// TwinCAT 3 PLC project tc_project_app
// ProgramVersion: 3.1.4023.0
// libraries:
//   Get_Nc_Error_Texts_and_descriptions, * (Beckhoff Automation GmbH & Co. KG)
//   Tc2_EtherCAT, * (Beckhoff Automation GmbH)
//   Tc2_MC2, * (Beckhoff Automation GmbH)
//   Tc2_Standard, * (Beckhoff Automation GmbH)
//   Tc2_SUPS, * (Beckhoff Automation GmbH)
//   Tc2_System, * (Beckhoff Automation GmbH)
//   Tc2_Utilities, * (Beckhoff Automation GmbH)
//   Tc3_MC2_AdvancedHoming, * (Beckhoff Automation GmbH)
//   Tc3_Module, * (Beckhoff Automation GmbH)
//   VisuDialogs, * (System)
//   Tc2_Math,3.3.1.0,Beckhoff Automation GmbH
//   VisuSymbols,3.5.10.0,System
// project tree:
//   DUTs/ E_Beamline.TcDUT, E_ResetZero.TcDUT, stFaultType.TcDUT, E_LightShutterSystemStates.TcDUT, E_SeqRangePosStates.TcDUT, E_NeutronFactoryStates.TcDUT, ST_LightShutter.TcDUT
//   / GlobalTextList.TcGTLO, PlcTask.TcTTO, PlcTaskCom.TcTTO, Visualization Manager.TcVMO (not stored)
//   GVLs/ GVL_APP.TcGVL
//   POUs/Application_Specific/Applications/ Application_Template.TcPOU, FB_ResetZero.TcPOU, HomeStepBlockDetection.TcPOU, NeutronFactoryStates.TcPOU, LightShutterSystemStates.TcPOU, SeqRangePos.TcPOU
//   POUs/Application_Specific/Axes/ Axis_Template.TcPOU, Pneumatics_Template.TcPOU
//   POUs/ MAIN.TcPOU
//   tc_mca_std_lib/DUTs/ E_AxisParameters.TcTLEO (not stored), E_HomingRoutines.TcTLEO (not stored), E_AxisParameters.TcTLEO (not stored), E_MotorTypeClass.TcDUT (not stored), E_EncoderTypeClass.TcDUT (not stored), E_HomeSwitchTypeClass.TcDUT (not stored), E_RestorePosition.TcDUT (not stored), E_SlitPairStates.TcDUT (not stored), ST_AxisConfig.TcDUT (not stored), ST_StepBlockConfig.TcDUT (not stored), ST_AxisControl.TcDUT (not stored), E_MotionFunctions.TcDUT (not stored), ST_AxisDescription.TcDUT (not stored), ST_AxisError.TcDUT (not stored), ST_AxisInputs.TcDUT (not stored), ST_AxisPersistent.TcDUT (not stored), ST_GearAxis.TcDUT (not stored), ST_AxisStatus.TcDUT (not stored), ST_AxisStruct.TcDUT (not stored)
//   tc_mca_std_lib/DUTs/Pneumatics/ E_PneumaticAxisErrors.TcDUT (not stored), E_PneumaticMode.TcDUT (not stored), ST_PneumaticAxisControl.TcDUT (not stored), ST_PneumaticAxisConfig.TcDUT (not stored), ST_PneumaticAxisInputs.TcDUT (not stored), ST_PneumaticAxisOutputs.TcDUT (not stored), ST_PneumaticAxisStatus.TcDUT (not stored), ST_PneumaticAxisStruct.TcDUT (not stored)
//   tc_mca_std_lib/GVLs/ GVL.TcGVL (not stored)
//   tc_mca_std_lib/POUs/Motion/ FB_Axis.TcPOU (not stored), FB_SlitPair.TcPOU (not stored)
//   tc_mca_std_lib/POUs/Motion/Homing/ FB_Homing.TcPOU (not stored)
//   tc_mca_std_lib/POUs/Pneumatics/ FB_PneumaticAxis.TcPOU (not stored)
//   tc_mca_std_lib/VISUs/ languageSupport.TcTLO (not stored), MainVisu.TcVIS (not stored), PneumaticsVisu.TcVIS (not stored), visuTextLinks.TcTLO (not stored)
//   tc_pils/tc_pils_app_specific/GVLs/ GVL_PILS.TcGVL
//   tc_pils/tc_pils_app_specific/POUs/ PILS_DEVICES.TcPOU
//   tc_pils/tc_pils_generic/DUTs/ E_Permission.TcDUT (not stored), E_PILS_ParamControl.TcDUT (not stored), E_PILS_ParamControlCmd.TcDUT (not stored), E_PILS_State.TcDUT (not stored), ST_1201.TcDUT (not stored), ST_1202.TcDUT (not stored), ST_1204.TcDUT (not stored), ST_1602.TcDUT (not stored), ST_5008.TcDUT (not stored), ST_5010.TcDUT (not stored), ST_AxisParameters.TcDUT (not stored), ST_DeviceInfo.TcDUT (not stored), ST_Indexer.TcDUT (not stored), ST_Indexer_InfoTyp0.TcDUT (not stored), ST_ParamOutput.TcDUT (not stored), U_IndexerData.TcDUT (not stored)
//   tc_pils/tc_pils_generic/POUs/ COMM.TcPOU (not stored)
//   tc_pils/tc_pils_generic/POUs/PILS_device_types/ FB_5010_Axis.TcPOU (not stored)
//   VISUs/ AcceleratorStates.TcVIS, languageTable.TcTLO, StepBlockDetection.TcVIS
// real-time tasks:
//   TASK PlcTask: cycle T#10ms, priority 10, ADS port 351
//   TASK PlcTaskCom: cycle T#2ms, priority 5, ADS port 350
// motion (NC):
//   TASK NC-Task 1 SAF: cycle T#2ms, priority 4, ADS port 501
//   TASK NC-Task 1 SVB: cycle T#10ms, priority 8, ADS port 511
//   AXIS Axis 1 (id 1)
//     Dynamic: AccelerationMaximum=1500, DecelerationMaximum=1500, Acceleration=50, Deceleration=50, Jerk=1000
//     Velo: RefSearch=10, RefSync=10, SlowManual=10, FastManual=15, Maximum=500
//     PositionAreaControl: Range=0.5
//     TargetPosControl: Range=0.5, Time=0.2
//     OtherSettings: AllowMotionCmdToSlave=true, PulseDistancePos=10, PulseDistanceNeg=10
//     encoder EncType=5
//       EncPara: ScaleFactorNumerator=60, ScaleFactorDenominator=4096, Inverse=true, ReferenceSystem=1
//         SoftEndMinControl: Range=1
//         SoftEndMaxControl: Range=500000
//         Inc: RefSoftSyncMask=#x0000ffff
//     drive DrvType=24
//       Analog: VeloReferenz=600, TorqueSetpointScale=10, ScaleFactorActTorque=0.1
//       TimeComp: TaskDelayCycles=1
//     controller CtrType=1
//       CtrPara: PriorControlFactor=1
//         PosDiffControl: Range=100
//         Observer: BandWidth=20
//   AXIS Axis 2 (id 2)
//     Dynamic: AccelerationMaximum=1500, DecelerationMaximum=1500, Acceleration=50, Deceleration=50, Jerk=1000
//     Velo: RefSearch=10, RefSync=10, SlowManual=10, FastManual=15, Maximum=500
//     PositionAreaControl: Range=0.5
//     TargetPosControl: Range=0.5, Time=0.2
//     OtherSettings: AllowMotionCmdToSlave=true, PulseDistancePos=10, PulseDistanceNeg=10
//     encoder EncType=5
//       EncPara: ScaleFactorNumerator=60, ScaleFactorDenominator=4096, Inverse=true, MaxCount=#xffffffff, ReferenceSystem=1
//         SoftEndMinControl: Range=1
//         SoftEndMaxControl: Range=500000
//         Inc: RefSoftSyncMask=#x0000ffff
//     drive DrvType=24
//       Analog: VeloReferenz=600, TorqueSetpointScale=10, ScaleFactorActTorque=0.1
//       TimeComp: TaskDelayCycles=1
//     controller CtrType=1
//       CtrPara: PriorControlFactor=1
//         PosDiffControl: Range=100
//         Observer: BandWidth=20
//   AXIS Axis 3 (id 3)
//     Dynamic: Acceleration=3439.33, Deceleration=3439.33, Jerk=10318
//     Velo: RefSearch=22.9288618666667, RefSync=22.9288618666667, SlowManual=114.644309333333, FastManual=687.865856, Fast=2292.88618666667, Maximum=2292.89
//     OtherSettings: AllowMotionCmdToSlave=true
//     encoder EncType=19
//       EncPara: ScaleFactorNumerator=104.8576, ScaleFactorDenominator=1048576, MaxCount=#xffffffff
//     drive DrvType=16
//       DrvPara: MaxCount=#xffffffff, DriveControlDWord=#x00020000
//         Analog: VeloReferenz=2522.17480533333, VeloScale=32, TorqueSetpointScale=10, ScaleFactorActTorque=0.1
//         TimeComp: TaskDelayCycles=1
//     controller CtrType=1
//       CtrPara: PriorControlFactor=1
//         PosDiffControl: Enable=false
//         Observer: BandWidth=20
// I/O:
//   DEVICE Device 1 (EtherCAT), AmsNetId 5.65.73.226.2.1
//     Term 1 (EK1200) [EK1200-5000 EtherCAT Power supply (2A E-Bus)]
//       Term 2 (EL1808) [EL1808 8Ch. Dig. Input 24V, 3ms]
//       Term 3 (EL2819) [EL2819 16Ch. Dig. Output 24V, 0,5A, Diagnostic]
//       Term 4 (EL5002) [EL5002 2Ch. SSI Encoder]
//       Term 5 (EL2014) [EL2014 4Ch. Dig. Output 24V, 0,5A, Diagnostic]
//       Term 6 (EL7041-0052) [EL7041-0052 1Ch. Stepper motor output stage (50V, 5A)]
//       Term 7 (EL7041-0052) [EL7041-0052 1Ch. Stepper motor output stage (50V, 5A)]
//       Term 8 (EL3204) [EL3204 4Ch. Ana. Input PT100 (RTD)]
//       Term 18 (EL7201) [EL7201 1Ch. MDP742 Servo motor output stage (50V, 4A)]
//       Term 9 (EL9011) [EL9011 End Terminal]
//   DEVICE Device 4 (COM Port)
// variable links:
//   (this object) <-> Device 1 (EtherCAT)/Term 1 (EK1200)/Term 4 (EL5002)
//     Enc/Inputs/In/nDataIn1 <-> SSI Inputs Channel 1/Counter value
//     Enc/Inputs/In/nDataIn1 <-> SSI Inputs Channel 2/Counter value
//     Enc/Inputs/In/nState1 <-> SSI Inputs Channel 1/Data error
//     Enc/Inputs/In/nState1 <-> SSI Inputs Channel 2/Data error
//     Enc/Inputs/In/nState1 @bit 3 <-> SSI Inputs Channel 1/Data mismatch
//     Enc/Inputs/In/nState1 @bit 3 <-> SSI Inputs Channel 2/Data mismatch
//     Enc/Inputs/In/nState1 @bit 1 <-> SSI Inputs Channel 1/Frame error
//     Enc/Inputs/In/nState1 @bit 1 <-> SSI Inputs Channel 2/Frame error
//     Enc/Inputs/In/nState1 @bit 2 <-> SSI Inputs Channel 1/Power failure
//     Enc/Inputs/In/nState1 @bit 2 <-> SSI Inputs Channel 2/Power failure
//     Enc/Inputs/In/nState2 @bit 5 <-> SSI Inputs Channel 1/Sync error
//     Enc/Inputs/In/nState2 @bit 5 <-> SSI Inputs Channel 2/Sync error
//     Enc/Inputs/In/nState2 @bit 6 <-> SSI Inputs Channel 1/TxPDO State
//     Enc/Inputs/In/nState2 @bit 6 <-> SSI Inputs Channel 2/TxPDO State
//     Enc/Inputs/In/nState2 @bit 7 <-> SSI Inputs Channel 1/TxPDO Toggle
//     Enc/Inputs/In/nState2 @bit 7 <-> SSI Inputs Channel 2/TxPDO Toggle
//     Enc/Inputs/In/nState4 @bit 1 <-> WcState/InputToggle
//     Enc/Inputs/In/nState4 <-> WcState/WcState
//   (this object) <-> Device 1 (EtherCAT)/Term 1 (EK1200)/Term 6 (EL7041-0052)
//     Drive/Inputs/In/nState1 @bit 3 <-> STM Status/Error
//     Drive/Inputs/In/nState1 @bit 5 <-> STM Status/Moving negative
//     Drive/Inputs/In/nState1 @bit 4 <-> STM Status/Moving positive
//     Drive/Inputs/In/nState1 @bit 1 <-> STM Status/Ready
//     Drive/Inputs/In/nState1 <-> STM Status/Ready to enable
//     Drive/Inputs/In/nState1 @bit 6 <-> STM Status/Torque reduced
//     Drive/Inputs/In/nState1 @bit 2 <-> STM Status/Warning
//     Drive/Inputs/In/nState2 @bit 3 <-> STM Status/Digital input 1
//     Drive/Inputs/In/nState2 @bit 4 <-> STM Status/Digital input 2
//     Drive/Inputs/In/nState2 @bit 5 <-> STM Status/Sync error
//     Drive/Inputs/In/nState2 @bit 7 <-> STM Status/TxPDO Toggle
//     Drive/Inputs/In/nState4 @bit 1 <-> WcState/InputToggle
//     Drive/Inputs/In/nState4 <-> WcState/WcState
//     Drive/Outputs/Out/nCtrl1 <-> STM Control/Enable
//     Drive/Outputs/Out/nCtrl1 @bit 2 <-> STM Control/Reduce torque
//     Drive/Outputs/Out/nCtrl1 @bit 1 <-> STM Control/Reset
//     Drive/Outputs/Out/nDataOut2[0] <-> STM Velocity/Velocity
//   (this object) <-> Device 1 (EtherCAT)/Term 1 (EK1200)/Term 7 (EL7041-0052)
//     Drive/Inputs/In/nState1 @bit 3 <-> STM Status/Status/Error
//     Drive/Inputs/In/nState1 @bit 5 <-> STM Status/Status/Moving negative
//     Drive/Inputs/In/nState1 @bit 4 <-> STM Status/Status/Moving positive
//     Drive/Inputs/In/nState1 @bit 1 <-> STM Status/Status/Ready
//     Drive/Inputs/In/nState1 <-> STM Status/Status/Ready to enable
//     Drive/Inputs/In/nState1 @bit 6 <-> STM Status/Status/Torque reduced
//     Drive/Inputs/In/nState1 @bit 2 <-> STM Status/Status/Warning
//     Drive/Inputs/In/nState2 @bit 3 <-> STM Status/Status/Digital input 1
//     Drive/Inputs/In/nState2 @bit 4 <-> STM Status/Status/Digital input 2
//     Drive/Inputs/In/nState2 @bit 5 <-> STM Status/Status/Sync error
//     Drive/Inputs/In/nState2 @bit 7 <-> STM Status/Status/TxPDO Toggle
//     Drive/Inputs/In/nState4 @bit 1 <-> WcState/InputToggle
//     Drive/Inputs/In/nState4 <-> WcState/WcState
//     Drive/Outputs/Out/nCtrl1 <-> STM Control/Control/Enable
//     Drive/Outputs/Out/nCtrl1 @bit 2 <-> STM Control/Control/Reduce torque
//     Drive/Outputs/Out/nCtrl1 @bit 1 <-> STM Control/Control/Reset
//     Drive/Outputs/Out/nDataOut2[0] <-> STM Velocity/Velocity
//   (this object) <-> Device 1 (EtherCAT)/Term 1 (EK1200)/Term 18 (EL7201)
//     Drive/Inputs/In/nDcOutputTime <-> InfoData/DcOutputShift
//     Drive/Inputs/In/nState1 <-> DRV Statusword/Statusword
//     Drive/Inputs/In/nState2 <-> DRV Statusword/Statusword @bit 8
//     Drive/Inputs/In/nState4 @bit 1 <-> WcState/InputToggle
//     Drive/Inputs/In/nState4 <-> WcState/WcState
//     Drive/Outputs/Out/nCtrl1 <-> DRV Controlword/Controlword
//     Drive/Outputs/Out/nCtrl2 <-> DRV Controlword/Controlword @bit 8
//     Drive/Outputs/Out/nDataOut2 <-> DRV Target velocity/Target velocity
//     Enc/Inputs/In/nDataIn1 <-> FB Position/Position
//     Enc/Inputs/In/nDcInputTime <-> InfoData/DcInputShift
//     Enc/Inputs/In/nState4 @bit 1 <-> WcState/InputToggle
//     Enc/Inputs/In/nState4 <-> WcState/WcState
//   tc_project_app Instance <-> Device 1 (EtherCAT)/Term 1 (EK1200)/Term 2 (EL1808)
//     PlcTaskCom Inputs/GVL.astAxes[1].stInputs.bHomeSensor <-> Channel 3/Input
//     PlcTaskCom Inputs/GVL.astAxes[2].stInputs.bHomeSensor <-> Channel 7/Input
//     PlcTaskCom Inputs/GVL.astAxes[1].stInputs.bLimitBwd <-> Channel 2/Input
//     PlcTaskCom Inputs/GVL.astAxes[2].stInputs.bLimitBwd <-> Channel 6/Input
//     PlcTaskCom Inputs/GVL.astAxes[1].stInputs.bLimitFwd <-> Channel 1/Input
//     PlcTaskCom Inputs/GVL.astAxes[2].stInputs.bLimitFwd <-> Channel 5/Input
//   tc_project_app Instance <-> Device 1 (EtherCAT)/Term 1 (EK1200)/Term 3 (EL2819)
//     PlcTaskCom Outputs/Axis_Template.bPowerSwitchesAxis1 <-> DIG Outputs/Channel 1/Output
//     PlcTaskCom Outputs/Axis_Template.bPowerSwitchesAxis2 <-> DIG Outputs/Channel 5/Output
//   tc_project_app Instance <-> Device 1 (EtherCAT)/Term 1 (EK1200)/Term 5 (EL2014)
//     PlcTask Outputs/Axis_Template.bPowerEncAxis1 <-> DIG Outputs/Channel 1/Output
//     PlcTask Outputs/Axis_Template.bPowerEncAxis2 <-> DIG Outputs/Channel 2/Output
//   tc_project_app Instance <-> NC-Task 1 SAF/Axes/Axis 1
//     PlcTask Inputs/GVL.astAxes[1].Axis.NcToPlc <-> Outputs/ToPlc
//     PlcTask Outputs/GVL.astAxes[1].Axis.PlcToNc <-> Inputs/FromPlc
//   tc_project_app Instance <-> NC-Task 1 SAF/Axes/Axis 2
//     PlcTask Inputs/GVL.astAxes[2].Axis.NcToPlc <-> Outputs/ToPlc
//     PlcTask Outputs/GVL.astAxes[2].Axis.PlcToNc <-> Inputs/FromPlc
//   tc_project_app Instance <-> NC-Task 1 SAF/Axes/Axis 3
//     PlcTask Inputs/GVL.astAxes[3].Axis.NcToPlc <-> Outputs/ToPlc
//     PlcTask Outputs/GVL.astAxes[3].Axis.PlcToNc <-> Inputs/FromPlc

CONFIGURATION tc_project_app
    RESOURCE PLC ON TwinCAT3
        TASK PlcTask(INTERVAL := T#10ms, PRIORITY := 10);
        TASK PlcTaskCom(INTERVAL := T#2ms, PRIORITY := 5);
        PROGRAM MAIN WITH PlcTask : MAIN;
        PROGRAM COMM WITH PlcTaskCom : COMM;
    END_RESOURCE
END_CONFIGURATION

// ---- DUTs/E_Beamline.TcDUT
{attribute 'qualified_only'}
{attribute 'strict'}
TYPE E_Beamline :
(
    Miracles := 1,
	Heimdal
);
END_TYPE

// ---- DUTs/E_ResetZero.TcDUT
{attribute 'qualified_only'}
{attribute 'strict'}
TYPE E_ResetZero :
(
    INIT := 0,
	HOME_AXIS,
	FIND_POS_ONE,
	PREPARE_POS_ONE_X,
	RECORD_POS_ONE_X,
	PREPARE_POS_ONE_Y,
	RECORD_POS_ONE_Y,
	FIND_POS_TWO,
	POSITIONING
);
END_TYPE

// ---- DUTs/stFaultType.TcDUT
TYPE stFaultType :
	STRUCT
		sFaultType	:	STRING(255);
	END_STRUCT
END_TYPE

// ---- DUTs/E_LightShutterSystemStates.TcDUT
{attribute 'qualified_only'}
{attribute 'strict'}
TYPE E_LightShutterSystemStates :
(
    Init := 0,
	ClosedOff,
	ClosedStandby,
	Opening,
	Open,
	OpenToOpen,
	Adjusting,
	ResetZero,
	Closing,
	Maintenance,
	SinglePortMaintenance_ClosedStandby,
	SinglePortMaintenance_Opening,
	SinglePortMaintenance_Open,
	SinglePortMaintenance_Closing,
	LSS_Maintenance,
	Fault	
);
END_TYPE

// ---- DUTs/E_SeqRangePosStates.TcDUT
{attribute 'qualified_only'}
{attribute 'strict'}
TYPE E_SeqRangePosStates :
(
    INIT := 0,
    CHECK_HOME_STATUS,
    HOME_MOTOR,
    CHECK_HOME_COMPLETE,
    MOTOR_OPERATIONAL,
	POS_ZERO,
	POS_ONE,
	POS_TWO,
	POSITIONING,
    CLEAR_CALIBRATION,
    ERROR,
    ERROR_RESET_AXES,
    ERROR_RESET_CHECK
);
END_TYPE

// ---- DUTs/E_NeutronFactoryStates.TcDUT
{attribute 'qualified_only'}
{attribute 'strict'}
TYPE E_NeutronFactoryStates :
(
    Disabled := 0,
	Maintenance,
	StartUp,
	CoolingDown,
	NotConfirmedReady,
	ConfirmedReady	
);
END_TYPE

// ---- DUTs/ST_LightShutter.TcDUT
(*These are axis parameters that are set up during commissioning and
in theory don't neeed to be change as part of daily moving of axes.
For instance they may be changed due to poor parameter selection
or change of instrument configuration.*)
TYPE ST_LightShutter :
STRUCT
	//name? beamline nbr?
	// Are we also to store closed position?
    // Add status of switches?
	nbrOfPos : USINT; // 1 or 2 foxal points
	curPosNbr : USINT := 1;
	pos : ARRAY[1..2] OF LREAL := [0,0];
	
END_STRUCT
END_TYPE

// ---- GVLs/GVL_APP.TcGVL
{attribute 'qualified_only'}
VAR_GLOBAL
	aPosSwitch : ARRAY[1..GVL_APP.nAXIS_NUM, 1..2] OF BOOL;
END_VAR

VAR_GLOBAL CONSTANT
    nAXIS_NUM: UINT := 3; (*~ (OPC: 1 : available for OPC-clients)
                         (OPC_PROP[0005]: 1 : OPC_PROP_RIGHTS, here read only) *)
    nPNEUMATIC_AXIS_NUM: UINT := 0;
END_VAR

VAR_GLOBAL PERSISTENT
	aLightShutters : ARRAY[1..GVL_APP.nAXIS_NUM] OF ST_LightShutter;
END_VAR

// ---- tc_pils/tc_pils_app_specific/GVLs/GVL_PILS.TcGVL
  VAR_GLOBAL
    sPLCName: STRING[34] := 'Crate_026';
    sPLCVersion: STRING[34] := '0.9.3';
    sPLCAuthor1: STRING[34] := 'tc_lab_mcu026.git';
    sPLCAuthor2: STRING[34] := 'ESS Lund';

//PILS Devices
//First available memory area for PILS devices is 104. 64-99 is used by the indexer
//Run the python script "check_fix_gvl_pils.py" to check that the PILS devices have a correct memory allocation

    //Axis #1                  Pils-device typ
    stMotorM1       AT %MB104: ST_5010;
    fbMotorM1: FB_5010_Axis := (nPILSDeviceNumber := 1);
    stMotorM1Param: ST_AxisParameters := (eMicrostepsPermission := E_Permission.eHidden,
                                          eResolutionPermission := E_Permission.eHidden,
                                          eAccelerationPermission := E_Permission.eWrite,
                                          eHomePositionPermission := E_Permission.eWrite,
                                          eHomingVelocityPermission := E_Permission.eWrite,
                                          eLagErrorPermission := E_Permission.eWrite,
                                          eTargetPositionWindowPermission := E_Permission.eWrite,
                                          eUserMaxPermission := E_Permission.eWrite,
                                          eUserMinPermission := E_Permission.eWrite,
                                          eVelocityPermission := E_Permission.eWrite,
                                          eSoftPosMinimumLimitEnablePermission := E_Permission.eWrite,
                                          eSoftPosMaximumLimitEnablePermission := E_Permission.eWrite,
                                          eHomeSequencePermission := E_Permission.eWrite,
                                          eEncoderScalingNumeratorPermission := E_Permission.eWrite,
                                          eEncoderScalingDenominatorPermission := E_Permission.eWrite,
                                          eMaximumVelocityPermission := E_Permission.eWrite);
										  
	//Axis #2                  Pils-device typ
    stMotorM2       AT %MB136: ST_5010;
    fbMotorM2: FB_5010_Axis := (nPILSDeviceNumber := 2);
    stMotorM2Param: ST_AxisParameters := (eMicrostepsPermission := E_Permission.eHidden,
                                          eResolutionPermission := E_Permission.eHidden,
                                          eAccelerationPermission := E_Permission.eWrite,
                                          eHomePositionPermission := E_Permission.eWrite,
                                          eHomingVelocityPermission := E_Permission.eWrite,
                                          eLagErrorPermission := E_Permission.eWrite,
                                          eTargetPositionWindowPermission := E_Permission.eWrite,
                                          eUserMaxPermission := E_Permission.eWrite,
                                          eUserMinPermission := E_Permission.eWrite,
                                          eVelocityPermission := E_Permission.eWrite,
                                          eSoftPosMinimumLimitEnablePermission := E_Permission.eWrite,
                                          eSoftPosMaximumLimitEnablePermission := E_Permission.eWrite,
                                          eHomeSequencePermission := E_Permission.eWrite,
                                          eEncoderScalingNumeratorPermission := E_Permission.eWrite,
                                          eEncoderScalingDenominatorPermission := E_Permission.eWrite,
                                          eMaximumVelocityPermission := E_Permission.eWrite);
										  
								
	stPowerSwitchesAxis1	AT %MB168: ST_1201;
	//fbMotorM2: FB_5010_Axis := (nPILSDeviceNumber := 2);
	//stPowerSwitchesAxis2	AT %MB170: ST_1201;
	stPowerSwitchesAxis2	AT %MB170: ST_1201;
	stPowerSwitchesAxis1Ctr AT %MB172: ST_1602;
	//stPowerSwitchesAxis2Ctr AT %MB176: ST_1602;
	

// Array of Devices
// Modify the array to fit the number of devices you have
// nUnit codes: mm = 16xfd04, degrees = 16x000C, Celsius =16x0009, Kelvin 16x0008

    astDevices: ARRAY [1..6] OF ST_DeviceInfo :=[ 									//axis specific.........generic
        (nTypCode := 16#5010, sName := 'M1 Lower', nOffset := 104, nUnit := 16#FD04, asAUX := [(''),(''),(''),(''),(''),(''),(''),(''),(''),(''),(''),(''),(''),(''),(''),(''),(''),('InterlockFwd'),('InterlockBwd'),('localMode'),('inTargetPos'),('homeSensor'),('notHomed'),('enabled')], nFlags := 1),
		(nTypCode := 16#5010, sName := 'M2 Higher', nOffset := 136, nUnit := 16#FD04, asAUX := [(''),(''),(''),(''),(''),(''),(''),(''),(''),(''),(''),(''),(''),(''),(''),(''),(''),('InterlockFwd'),('InterlockBwd'),('localMode'),('inTargetPos'),('homeSensor'),('notHomed'),('enabled')], nFlags := 1),
		(nTypCode := 16#1201, sName:= 'bPowerSwitchesAxis#1', nOffset := 168),
		(nTypCode := 16#1201, sName:= 'bPowerSwitchesAxis#2', nOffset := 170),
		(nTypCode := 16#1602, sName:= 'bPowerSwitchesAxisCtr#1', nOffset := 172)
		//(nTypCode := 16#1602, sName:= 'bPowerSwitchesAxisCtr#2', nOffset := 176)
		];
END_VAR

// ---- POUs/MAIN.TcPOU
PROGRAM MAIN
VAR
    sVersion: STRING := '1.0.0';
    afbAxes: ARRAY [1..GVL_APP.nAXIS_NUM] OF FB_Axis;
    afbPneumaticAxes: ARRAY [1..GVL_APP.nPNEUMATIC_AXIS_NUM] OF FB_PneumaticAxis;
    hmiAxisSelection: INT := 1; //Not possible to use local hmi variables for array indexes
    hmiPneumaticAxisSelection: INT := 1;
//Startup, Shutdown and UPS
    fbUPS: FB_S_UPS_CX51x0;
    eUpsMode: E_S_UPS_Mode := eSUPS_WrPersistData_Shutdown;
    eStartUp: (eColdStart, eReadAxisFeedbackType, eCheckReadDone, eExecuteRestore, eCheckRestore, eFinishRestore);
    bPositionRestoreDone: BOOL := FALSE;
    bRestoreExecute: BOOL := FALSE;
    bExecuteReadEncRefSys: BOOL := FALSE;
    nRetry: INT;
    iAxes : UINT; //index for for loops in Position recovery actions
    afbReadEncRefSys: ARRAY [1..GVL_APP.nAXIS_NUM] OF MC_ReadParameter;
    afbRestorePosition: ARRAY [1..GVL_APP.nAXIS_NUM] OF MC_SetPosition;
    fbGetDeviceIdentification: FB_GetDeviceIdentificationEx;
END_VAR

VAR PERSISTENT
    bRestoreOnStartup: BOOL;
END_VAR

POSITION_RECOVERY();
AXES();
PROG();

ACTION AXES:
//Get task index for Axes parameters initialization.
GVL.fbGetCurTaskIndex();

//Create an stAxisStruct for every axis in the project.
FOR GVL.iAxis := 1 TO GVL_APP.nAXIS_NUM DO
    afbAxes[GVL.iAxis](stAxisStruct := GVL.astAxes[GVL.iAxis]);
END_FOR

FOR GVL.iPneumaticAxis := 1 TO GVL_APP.nPNEUMATIC_AXIS_NUM DO
    afbPneumaticAxes[GVL.iPneumaticAxis](stPneumaticAxisStruct := GVL.astPneumaticAxes[GVL.iPneumaticAxis]);
END_FOR
END_ACTION

ACTION CHECK_UPS:
fbUPS(eUpsMode := eUpsMode);

IF eGlobalSUpsState = eSUPS_PowerFailure THEN
    //first cycle of powerfailure
    //execute code that should only be done once with each powerfailure, i.e. increase powerfailure counter
    bRestoreOnStartup := TRUE;
    STORE_PERSISTENT();
    RETURN;
ELSIF eGlobalSUpsState <> eSUPS_PowerOK THEN
    //next cycles of powerfailure
    //skip regular code execution for the remaining cycles of the powerfailure/writing of persistent data/quick shutdown...
    RETURN;
END_IF
END_ACTION

ACTION POSITION_RECOVERY:
fbGetDeviceIdentification(bExecute := TRUE);
IF (fbGetDeviceIdentification.stDevIdent.strHardwareSerialNo <> '0') THEN
    CHECK_UPS();
    RESTORE_POSITIONS();
END_IF
END_ACTION

ACTION PROG:
//Call the programs that are defined in the "Application Specific" folder.
//Create as many programs in that folder as axes and applications you have or need

//Axes program calls
Axis_Template();
Pneumatics_Template();

//Application program calls
Application_Template();
//SeqRangePos();
//NeutronFactoryStates();

//LightShutterSystemStates();
HomeStepBlockDetection();
END_ACTION

ACTION RESTORE_POSITIONS:
//This ACT will restore the position of an incremental axis on startup with the act position it read before losing power.
//It checks the type of axis, 0=incremental, and that the axis was stationary at shut down.
//Because 0 equates to incremental we also need to check that the data is valid, otherwise by default it would restore all axes.
//By default an axis will not restore the position unless it is set to opt-in, i.e. GVL.aAxes[iAxes].stConfig.eRestorePosition is non-zero.
//This needs to be initialised somewhere in TwinCAT code otherwise it will not be available at start up.
//A restore will only be performed on a loss of power, this code shouldn't make any changes on a reset cold, a rest origin or a download.
//There is a enum to allow for different types of restore modes, currently only one is implemented.
//0 'DontRestore'
//1 'RestoreWithoutHome' -restores the position using a set position fb and does not set the home bit in the axis struct.
//Note from Beckhoff: "A maximum of 1 MB persistent data can be reliably saved over the entire service life."

IF bRestoreOnStartup AND eGlobalSUpsState = eSUPS_PowerOK THEN
    bRestoreOnStartup := FALSE;
    bRestoreExecute := TRUE;
END_IF

//Upon startup bPositionRestoreDone will be set to FALSE, after successfully completing the following code it will be set TRUE
//and should stay TRUE for the rest of the time the PLC is operational, thus this routine should only be completed once.
IF bRestoreExecute AND NOT bPositionRestoreDone THEN
    //Cycle through function blocks that read the encoder reference system i.e. whether axis is incremental or absolute
    //Result stored in Value, 0=Inc 1=Abs, execute set during the case statement
    FOR iAxes := 1 TO GVL_APP.nAXIS_NUM DO
        afbReadEncRefSys[iAxes](
          Axis := GVL.astAxes[iAxes].Axis,
          Enable := bExecuteReadEncRefSys,
          ParameterNumber := MC_AxisParameter.AxisEncoderReferenceSystem,
          ReadMode := E_READMODE.READMODE_ONCE);
    END_FOR

    //Cycle through set position function blocks for each axis
    FOR iAxes := 1 TO GVL_APP.nAXIS_NUM DO
        afbRestorePosition[iAxes](
         Axis := GVL.astAxes[iAxes].Axis,
         Position := astAxesPersistent[iAxes].fPositionAtShutdown);
    END_FOR

    CASE eStartUp OF
        eColdStart:
        //First cycle of the PLC, do nothing just give one cycle for variables to initialise
            IF NOT bPositionRestoreDone THEN
                eStartUp := eReadAxisFeedbackType;
                nRetry := 0;
            END_IF

        eReadAxisFeedbackType:
        //Exectute the function blocks to read the encoder reference system (0=inc OR 1=ABS)
            bExecuteReadEncRefSys := TRUE;
            eStartUp := eCheckReadDone;

        eCheckReadDone:
        //Check the encoder reference system has been read for all axis -> if busy then continue with PLC cycle and check again next time.
        //If afbReadEncRefSys not started then go back a step.
        //If any axes result in an error the code will get stuck here, this happens if GVL_APP.nAXIS_NUM is not set correctly
            FOR iAxes := 1 TO GVL_APP.nAXIS_NUM DO
                IF afbReadEncRefSys[iAxes].Valid = FALSE THEN
                    IF afbReadEncRefSys[iAxes].Busy = TRUE THEN
                        //Exit MAIN.STARTUP Action and wait till next cycle, needs to cycle through whole program in order for data to update
                        RETURN;
                    ELSE
                        //Sometimes the code gets here and the afbReadEncRefSys[iAxes] misses the rising edge. If  the code gets here it means
                        //valid=FALSE and .busy=FALSE which indicateds the FB probably hasn't started and thus needs to see a rising edge.
                        //Set execute to low, Exit MAIN.STARTUP and go back a step in the CASE statement.
                        bExecuteReadEncRefSys := FALSE;
                        eStartUp := eReadAxisFeedbackType;
                        nRetry := nRetry + 1; //counter used for troubleshooting to see how many cycles it takes before afbReadEncRefSys function blocks are read correctly
                        RETURN;
                    END_IF
                END_IF
            END_FOR
            //If the code gets here all axes either have .valid=TRUE for all axes
            eStartUp := eExecuteRestore;

        eExecuteRestore:
        //Execute position restore by setting afbRestorePosition.execute = TRUE
            FOR iAxes := 1 TO GVL_APP.nAXIS_NUM DO
                IF afbReadEncRefSys[iAxes].Valid = TRUE AND afbReadEncRefSys[iAxes].Value = 0 AND NOT(astAxesPersistent[iAxes].bMovingAtShutdown) THEN
                    IF GVL.astAxes[iAxes].stConfig.eRestorePosition = E_RestorePosition.eRestoreWithoutHome THEN
                        afbRestorePosition[iAxes].Execute := TRUE;
                    END_IF
                END_IF
            END_FOR
            eStartUp := eCheckRestore;

        eCheckRestore:
        //Check the set position fbs are finished
        //Nothing actually happens if the restore is not done, the code just returns from here each cycle and the
        //bPositionRestoreDone will never get set to TRUE and will take up cycle time
            FOR iAxes := 1 TO GVL_APP.nAXIS_NUM DO
                IF afbReadEncRefSys[iAxes].Valid = TRUE AND afbReadEncRefSys[iAxes].Value = 0 AND NOT(astAxesPersistent[iAxes].bMovingAtShutdown) THEN
                    IF GVL.astAxes[iAxes].stConfig.eRestorePosition = E_RestorePosition.eRestoreWithoutHome THEN
                        IF NOT afbRestorePosition[iAxes].Done THEN
                            RETURN;
                        END_IF
                    END_IF
                END_IF
            END_FOR
            eStartUp := eFinishRestore;

        eFinishRestore:
        //Remove execute = TRUE for afbRestorePosition
            FOR iAxes := 1 TO GVL_APP.nAXIS_NUM DO
                afbRestorePosition[iAxes].Execute := FALSE;
            END_FOR
            bPositionRestoreDone := TRUE;
            bRestoreExecute := FALSE;
    END_CASE
END_IF
END_ACTION

ACTION STORE_PERSISTENT:
FOR iAxes := 1 TO GVL_APP.nAXIS_NUM DO
    astAxesPersistent[iAxes].fPositionAtShutdown := GVL.astAxes[iAxes].Axis.NcToPlc.ActPos;
    IF GVL.astAxes[iAxes].Axis.NcToPlc.ActVelo <> 0 THEN
        astAxesPersistent[iAxes].bMovingAtShutdown := TRUE;
    ELSE
        astAxesPersistent[iAxes].bMovingAtShutdown := FALSE;
    END_IF
    astAxesPersistent[iAxes].bMovingAtShutdown := astAxesPersistent[iAxes].bMovingAtShutdown OR GVL.astAxes[iAxes].Axis.Status.Moving;
END_FOR
END_ACTION

END_PROGRAM

// ---- POUs/Application_Specific/Axes/Axis_Template.TcPOU
PROGRAM Axis_Template
VAR
//Outputs: Power for Limit switches, Home Sensors, etc.
    bPowerSwitchesAxis1 AT %Q*: BOOL:= TRUE;
    bPowerSwitchesAxis2 AT %Q*: BOOL:= TRUE;
	bPowerEncAxis1 AT %Q*: BOOL:=TRUE;
	bPowerEncAxis2 AT %Q*: BOOL:=TRUE;
	
//Hardware interlocks
    //bInterlockFwdOK AT %I*: BOOL;
	
END_VAR

//Axis_Template.bPowerSwitchesAxis1:=INT_TO_BOOL(GVL_PILS.stPowerSwitchesAxis1Ctr.nTargetValue);  //allows EPICS to control

//Initial parameters of an Axis
(*IF _TaskInfo[fbGetCurTaskIndex.index].FirstCycle THEN
    //Initial default values:
    GVL.astAxes[1].stConfig.eHomeSeq := 0;
    GVL.astAxes[1].stConfig.fHomePosition := 0.0;
    GVL.astAxes[1].stConfig.fHomeFinishDistance := 0.0;
END_IF*)

//Define ACTIONS() or write exclusive code for an specific axis.
(*Eg. Stop when temperature reaches certain values, reduce speed if  a signal is activated, etc.
Eg. GVL.astAxes[x].stControl.bInterlockFwd := NOT bInterlockFwdOK;*)

END_PROGRAM

// ---- POUs/Application_Specific/Axes/Pneumatics_Template.TcPOU
PROGRAM Pneumatics_Template
VAR
END_VAR

//Test the program to control pneumatic acutator through PneumaticsVisu.
//Currently implemented control of single solenoid through PLC and and manually, with two momentary push buttons.

END_PROGRAM

// ---- POUs/Application_Specific/Applications/Application_Template.TcPOU
PROGRAM Application_Template
VAR
//Define all necessary variables for your application
END_VAR

//Program any specific code or safety code for an specific application when it involves multiple axes
//Eg. Collision avoidance, interlocks, sequencing, etc.

END_PROGRAM

// ---- POUs/Application_Specific/Applications/HomeStepBlockDetection.TcPOU
PROGRAM HomeStepBlockDetection
VAR
	bJog : BOOL;
	bHome : BOOL;
	bFirst : BOOL := FALSE;
	nState : DINT := 0;
	
END_VAR

GVL.astAxes[3].stInputs.bLimitBwd := TRUE;
GVL.astAxes[3].stInputs.bLimitFwd := TRUE;

IF NOT bFirst THEN
	actInit();
END_IF

ACTION actInit:
GVL.astAxes[3].stConfig.stStepBlock.tDetectionVelocityTime := T#200MS;
GVL.astAxes[3].stConfig.stStepBlock.fAcceleration := 100;
GVL.astAxes[3].stConfig.stStepBlock.fDeceleration := 100;
GVL.astAxes[3].stConfig.stStepBlock.fDetectionVelocityLimit := GVL.astAxes[3].stConfig.fHomingVelFromCam*0.1;
GVL.astAxes[3].stConfig.stStepBlock.fDistanceLimit := 100000;
GVL.astAxes[3].stConfig.stStepBlock.fTorqueLimit := 50000000000000000;
GVL.astAxes[3].stConfig.stStepBlock.fTorqueTolerance := 50000000000000000;
GVL.astAxes[3].stConfig.stStepBlock.fVeloMax := GVL.astAxes[3].stConfig.fHomingVelFromCam;
GVL.astAxes[3].stConfig.stStepBlock.tTimeLimit := T#20000MS;


// Problematic to detect velocity correctly with stepper motor, is it possible?
// On the crates the connection between the motor axis and the linear rubber band
// seems to jump, which translates to that the shaft of the motor is not reduced in
// its velocity.
GVL.astAxes[1].stConfig.stStepBlock.tDetectionVelocityTime := T#60MS;
GVL.astAxes[1].stConfig.stStepBlock.fAcceleration := 100;
GVL.astAxes[1].stConfig.stStepBlock.fDeceleration := 100;
GVL.astAxes[1].stConfig.stStepBlock.fDetectionVelocityLimit := GVL.astAxes[3].stConfig.fHomingVelFromCam*0.007;
GVL.astAxes[1].stConfig.stStepBlock.fDistanceLimit := 100000;
GVL.astAxes[1].stConfig.stStepBlock.fTorqueLimit := 100;
GVL.astAxes[1].stConfig.stStepBlock.fTorqueTolerance := 100;
GVL.astAxes[1].stConfig.stStepBlock.fVeloMax := GVL.astAxes[3].stConfig.fHomingVelFromCam*0.01;
GVL.astAxes[1].stConfig.stStepBlock.tTimeLimit := T#20000MS;
END_ACTION

END_PROGRAM

// ---- POUs/Application_Specific/Applications/FB_ResetZero.TcPOU
FUNCTION_BLOCK FB_ResetZero

VAR_INPUT
	axisNbr : UINT;
	bAxisDone : BOOL;
END_VAR

VAR_OUTPUT
END_VAR

VAR
	usCurrentPos : USINT;
	eResetZeroInternal: E_ResetZero := E_ResetZero.INIT;
	fPosX : LREAL;
	fPosY : LREAL;
	fPosFocal : LREAL;
    TON_delayDone : TON;
END_VAR

VAR_IN_OUT
	bResetZero : BOOL;
	//bAxisDelayDone : BOOL;
END_VAR

TON_delayDone(IN:=bAxisDone, PT:=T#1S);

CASE eResetZeroInternal OF
			
	E_ResetZero.INIT:
		
		GVL.astAxes[axisNbr].stControl.bEnable := TRUE;
		usCurrentPos := 1; // Help variable for looping through first and if available, second, position
		
		IF GVL.astAxes[axisNbr].stStatus.bEnabled THEN
			eResetZeroInternal := E_ResetZero.HOME_AXIS;
		END_IF
		
	E_ResetZero.HOME_AXIS:
		// CHANGE to HomeByTorque and at top position.
		GVL.astAxes[axisNbr].stConfig.eHomeSeq := E_HomingRoutines.eHomeToLimit_Bwd;
		GVL.astAxes[axisNbr].stControl.eCommand := E_MotionFunctions.eHome;
		GVL.astAxes[axisNbr].stControl.bExecute := TRUE;				
		
		IF GVL.astAxes[axisNbr].stStatus.bDone AND NOT(GVL.astAxes[axisNbr].stInputs.bLimitBwd) THEN
			eResetZeroInternal := E_ResetZero.FIND_POS;
		END_IF
	
	E_ResetZero.FIND_POS:
		GVL.astAxes[axisNbr].stControl.eCommand:=E_MotionFunctions.eJog;
		// Can prob. not use bHomeSensor later. But other I/O LS - change direction also since zero at top?
		GVL.astAxes[axisNbr].stControl.bJogFwd:= NOT(GVL_APP.aPosSwitch[axisNbr, usCurrentPos]);
		
		IF GVL.astAxes[axisNbr].stStatus.bDone AND GVL_APP.aPosSwitch[axisNbr, usCurrentPos] THEN
			eResetZeroInternal := E_ResetZero.PREPARE_POS_X;
		END_IF
		
	E_ResetZero.PREPARE_POS_X:
		GVL.astAxes[axisNbr].stControl.bJogBwd:= GVL_APP.aPosSwitch[axisNbr, usCurrentPos];
		
		IF GVL.astAxes[axisNbr].stStatus.bDone AND NOT(GVL_APP.aPosSwitch[axisNbr, usCurrentPos]) THEN
			eResetZeroInternal := E_ResetZero.RECORD_POS_X;
		END_IF
		
	E_ResetZero.RECORD_POS_X:
		GVL.astAxes[axisNbr].stControl.fVelocity := 1;
		GVL.astAxes[axisNbr].stControl.bJogFwd := NOT(GVL_APP.aPosSwitch[axisNbr, usCurrentPos]);
		
		IF GVL.astAxes[axisNbr].stStatus.bDone AND GVL_APP.aPosSwitch[axisNbr, usCurrentPos] THEN
			fPosX := GVL.astAxes[axisNbr].stStatus.fActPosition;
			eResetZeroInternal := E_ResetZero.PREPARE_POS_Y;
		END_IF
		
	E_ResetZero.PREPARE_POS_Y:
		
		GVL.astAxes[axisNbr].stControl.fVelocity := GVL.astAxes[axisNbr].stConfig.fVelocityDefaultSlow;
		GVL.astAxes[axisNbr].stControl.bJogFwd := GVL_APP.aPosSwitch[axisNbr, usCurrentPos];
		
		IF GVL.astAxes[axisNbr].stStatus.bDone AND NOT(GVL_APP.aPosSwitch[axisNbr, usCurrentPos]) THEN
			eResetZeroInternal := E_ResetZero.RECORD_POS_Y;
		END_IF
		
	E_ResetZero.RECORD_POS_Y:
		GVL.astAxes[axisNbr].stControl.bJogBwd := NOT(GVL_APP.aPosSwitch[axisNbr, usCurrentPos]);
		
		IF GVL.astAxes[axisNbr].stStatus.bDone AND GVL_APP.aPosSwitch[axisNbr, usCurrentPos] THEN
		
			fPosY := GVL.astAxes[axisNbr].stStatus.fActPosition;
			fPosFocal := (fPosX+fPosY)/2;
			GVL_APP.aLightShutters[axisNbr].pos[usCurrentPos] := fPosFocal;
			
			// Check if axis has two position, then if not at pos two, go find it, otherwise quit.
			IF GVL_APP.aLightShutters[axisNbr].nbrOfPos = usCurrentPos THEN
				eResetZeroInternal := E_ResetZero.POSITIONING;
			ELSE
				usCurrentPos := usCurrentPos + 1;
				eResetZeroInternal := E_ResetZero.FIND_POS;
			END_IF
				
		END_IF
	
	E_ResetZero.POSITIONING:
		GVL.astAxes[axisNbr].stControl.eCommand := E_MotionFunctions.eMoveAbsolute;
		GVL.astAxes[axisNbr].stControl.fPosition := GVL_APP.aLightShutters[axisNbr].pos[GVL_APP.aLightShutters[axisNbr].curPosNbr];
		GVL.astAxes[axisNbr].stControl.bExecute := TRUE;
		
		IF TON_delayDone.Q THEN
			bResetZero := FALSE;
		END_IF
END_CASE
				
IF NOT bResetZero THEN // Transitioning from state - need to check axis status? 
	GVL.astAxes[axisNbr].stControl.bEnable := FALSE;
	eResetZeroInternal := E_ResetZero.INIT;
	//eLightShutterSystemState := E_LightShutterSystemStates.Open; // What should happen here?
END_IF

END_FUNCTION_BLOCK

// ---- POUs/Application_Specific/Applications/NeutronFactoryStates.TcPOU
PROGRAM NeutronFactoryStates
VAR
//Define all necessary variables for your application
	eNeutronFactoryState: E_NeutronFactoryStates := E_NeutronFactoryStates.Disabled;
END_VAR

CASE eNeutronFactoryState OF
	
	E_NeutronFactoryStates.Disabled:
		GVL.astAxes[MAIN.hmiAxisSelection].stControl.bEnable := FALSE;
	
	
	E_NeutronFactoryStates.Maintenance:
		GVL.astAxes[MAIN.hmiAxisSelection].stControl.bEnable := FALSE;
	
	
	E_NeutronFactoryStates.StartUp:
		GVL.astAxes[MAIN.hmiAxisSelection].stControl.bEnable := FALSE;
	
	
	E_NeutronFactoryStates.CoolingDown:
		GVL.astAxes[MAIN.hmiAxisSelection].stControl.bEnable := FALSE;
	
	
	E_NeutronFactoryStates.NotConfirmedReady:
		GVL.astAxes[MAIN.hmiAxisSelection].stControl.bEnable := FALSE;
	
	
	E_NeutronFactoryStates.ConfirmedReady:
		GVL.astAxes[MAIN.hmiAxisSelection].stControl.bEnable := TRUE;
		
END_CASE

END_PROGRAM

// ---- POUs/Application_Specific/Applications/LightShutterSystemStates.TcPOU
PROGRAM LightShutterSystemStates

VAR CONSTANT
	nAXIS_NUM : UINT := GVL_APP.nAXIS_NUM - 1; // JUST FOR TESTCRATE!
END_VAR

VAR
	eNeutronFactoryState: E_NeutronFactoryStates := E_NeutronFactoryStates.Disabled;
	// eResetZeroInternal: E_ResetZero := E_ResetZero.INIT;
	eLightShutterSystemState: E_LightShutterSystemStates := E_LightShutterSystemStates.Init;

	i   :   UINT:=0;
	
	bAxesDone: BOOL := FALSE; // Output variable of checkAxesDone
	bAxesHomed: BOOL := FALSE; // Output variable of checkVirtualHomed
	bInPos: BOOL; // Output variable of checkPos
	
	bNeutronFactory_Maintenance: BOOL;	// ?
	bMaintenancePermission: BOOL; 		// ?
	bMaintencancePerformed: BOOL;		// ?
	
	bStartup : BOOL := TRUE;	// Help var for indicating first cycle. Set to FALSE thereafter.
	bEnablePower: BOOL; 		// Input var for actCascadePower - COULD POWER BE INCLUDED IN ST_LightShutter?
	aDisabled: ARRAY [1..nAXIS_NUM] OF BOOL; // INCLUDE IN ST_LightShutter?
	
	bClosedShutters: BOOL := FALSE; // Output variable of checkClosedLimitSwitches
	bAllDisabled: BOOL := FALSE; // Output variable of checkAllDisabled
	
	// For Error Text
	//FaultType   :   stFaultType;
	//sErrorText : T_MaxString := '';
	//sErrorTextNc : T_MaxString := '';
	//strErrorText : DUT_ErrorText;
	//fbRead : FB_ReadTcNcErrorAndDescription;
	
	bLSSOpen: BOOL;		// Simulated signal, normally received from EPICS, to open/close shutters.
	bPSSPower: BOOL; 	// Simulated signal, normally received from EPICS letting us know that PSS has powered our drives.
	
	bOpenHiFake : BOOL; // Simulating a pos switch. To be replaced with physical switch.
	
	aOpenToOpen : ARRAY[1..nAXIS_NUM] OF BOOL; 	// Array of axes call to OpenToOpen
	aTON_delayOpenToOpen : ARRAY[1..nAXIS_NUM] OF TON;
	
	aResetZero : ARRAY[1..nAXIS_NUM] OF BOOL; 	// Array of axes call to ResetZero
	aFbResetZero : ARRAY[1..nAXIS_NUM] OF FB_ResetZero;
	
	aJogF : ARRAY[1..nAXIS_NUM] OF BOOL; 		// Array of axes call to Adjust
	aJogB : ARRAY[1..nAXIS_NUM] OF BOOL;		// Array of axes call to Adjust
	aTOF_delayDisable : ARRAY[1..nAXIS_NUM] OF TOF;
	aTON_delayDone : ARRAY[1..nAXIS_NUM] OF TON; // Remove - moved to FB_ResetZero
	
END_VAR

VAR PERSISTENT
	//aLightShutters : ARRAY[1..GVL_APP.nAXIS_NUM] OF ST_LightShutter;
END_VAR

actRunMethods(); // Update status

// Gets description of error codes and keeps them in mem --- IMPLEMENT ---
prgReadTcNcErrorAndDescription();

// Simulates position switch of second focal point
bOpenHiFake := GVL.astAxes[2].stStatus.fActPosition > 85 AND GVL.astAxes[2].stStatus.fActPosition < 100; 

actFaults(); 			// Checks errors --- IMPLEMENT ---

actPositionSwitches();	// Update GVL_APP.aPosSwitch with value of position switches
actDelayDisable(); 		// aTOF_delayDisable - Delay disabling of the drive of each axis
actDelayOpenToOpen();	// aTON_delayOpenToOpen - Delay OpenToOpen for each axis - for exit condition of actOpenToOpen
actDelayDone(); 		// aTON_delayDone - Delay done for each axis for handling e.g. exit conditions

//// To be mapped to EPICS signal. During tests mapped to DI. /////
IF NOT (eNeutronFactoryState = E_NeutronFactoryStates.Disabled) THEN
	bPSSPower := TRUE;
ELSE
	bPSSPower := FALSE;	
END_IF 
//////////////////////////

// Could also run a general actPower() here, and only set a boolean in the state machine
// true or not. This would also include a check if the device is disabled or if a specific
// axis demands control. Maybe a general bool if power is allowed or not should be given
// true or false in each state. Thus, if axis one requests power, but we are in closed off,
// nothing will happen.

// Dealing with race condition:
// 		Either TON and then check in IF --- This method is mainly used here.
// 		OR new state: POSITIONING_ WAITING
// 		OR while loop
//		COULD R_TRIG be used?

IF bStartup THEN 		// First cycle setup - _TaskInfo[1].FirstCycle did not work, why?)
	bStartup := FALSE;	// This IF will only be entered if it is the very first cycle.
	actInitAxis();
	// Currently resore only works for incremental encoder, not resolver. Easy fix.
	//GVL.astAxes[1].stConfig.eRestorePosition := 1; 
END_IF

CASE eLightShutterSystemState OF

	E_LightShutterSystemStates.Init:
		// Which should be the first state?
		// Need a manual config state which is to be used during commisionning.

		// The homing should be performed in the RESET substate of OPEN	
		// Maybe a requirement of being able to enter in the closed standby state 
		// should be to first have homed everything manually? Alternatively,
		// If not homed, the movement to first open could be performed by jogging
		// until hitting the position switch.
		// Homing in commisioning?

		bEnablePower := TRUE;
		actCascadePower();
		actCascadeHoming();

		IF _TaskInfo[1].CycleCount > 10000 AND bAxesHomed THEN
			eLightShutterSystemState := E_LightShutterSystemStates.ClosedOff;
			eNeutronFactoryState := E_NeutronFactoryStates.Disabled;
		END_IF		


	E_LightShutterSystemStates.ClosedOff:
		// All shutters closed, motor power off, brake on.
		// To do: LS verification and fault handling.

		bEnablePower := FALSE;
		actCascadePower();

		IF bLSSOpen AND bAxesDone THEN
			eNeutronFactoryState := E_NeutronFactoryStates.StartUp;
			eLightShutterSystemState := E_LightShutterSystemStates.ClosedStandby;
		END_IF

		IF bNeutronFactory_Maintenance THEN
			eLightShutterSystemState := E_LightShutterSystemStates.Maintenance;
		END_IF


	E_LightShutterSystemStates.ClosedStandby:
		// Verification of all shutters closed, motor power on (From PSS?), brake on.
		// To do: LS verification and fault handling.

		bEnablePower := FALSE;
		actCascadePower();

		IF bLSSOpen THEN
			eLightShutterSystemState := E_LightShutterSystemStates.Opening;
			eNeutronFactoryState := E_NeutronFactoryStates.NotConfirmedReady;
		END_IF

		IF NOT bLSSOpen AND bClosedShutters THEN
			eLightShutterSystemState := E_LightShutterSystemStates.ClosedOff;
			eNeutronFactoryState := E_NeutronFactoryStates.Disabled;
		END_IF


	E_LightShutterSystemStates.Opening:
		// Resolver monitoring of shutter pos. LSS monitor time for event to happen.
		// Motor power on. Brake off
		// To do: Fault handling. Time monitoring. 

		bEnablePower := TRUE;
		actCascadePower();
		actCascadeOpening();

		IF bAxesDone AND bInPos AND (NOT bClosedShutters OR bAllDisabled) THEN 
			// Also check bLSSOpen to be able to cancel Opening?
			// Also check positions?

			bEnablePower := FALSE;
			actCascadePower();
			eLightShutterSystemState := E_LightShutterSystemStates.Open; // Before transitioning, check NF?
			eNeutronFactoryState := E_NeutronFactoryStates.ConfirmedReady; // Not needed for us - or needed if to confirm "Open"?
		END_IF


	E_LightShutterSystemStates.Open:
		// Verification of all shutters open. Motor power off.
		// Brake on. (Dependent of specific OPEN TO OPEN pos)
		// To do: LS verification and fault handling.
		// Once inside here we allow individual shutter control.

		actPower();
		actOpenToOpen();
		actResetZero();		
		actJog();

		// Possibly create FB_LightShutter and add in array or structure
		// call it from here like:
		// for ... 
		// 		aLightShutter[i].fb_LightShutter(aOpenToOpen, aJogF/aJogB, aResetToZero)

		(*
		IF bJogB OR bJogF AND bLSSOpen THEN
			eLightShutterSystemState := E_LightShutterSystemStates.Adjusting;
			// fJogVelocity bug to be fixed in tc_mca_std_lib
			GVL.astAxes[MAIN.hmiAxisSelection].stControl.fJogVelocity := GVL.astAxes[MAIN.hmiAxisSelection].stConfig.fVelocityDefaultSlow*0.1;
			GVL.astAxes[MAIN.hmiAxisSelection].stControl.bEnable := TRUE;
		END_IF*)

		(*
		IF bOpenToOpen AND bLSSOpen THEN
			eLightShutterSystemState := E_LightShutterSystemStates.OpenToOpen;
			//fbOpenToOpen(bAxisDelayPower := bAxisDelayPower, bAxisDelayDone:= bAxisDelayDone);

		END_IF

		IF bResetZero AND bLSSOpen THEN // Use with AX drive - Torque homing.
			eLightShutterSystemState := E_LightShutterSystemStates.ResetZero;
		END_IF
		*)

		IF NOT bLSSOpen THEN
			eNeutronFactoryState := E_NeutronFactoryStates.CoolingDown;
			eLightShutterSystemState := E_LightShutterSystemStates.Closing;
		END_IF

	// Remove?
	E_LightShutterSystemStates.OpenToOpen: // Alt: Remove substate and have as option in Open instead
		// Substate of OPEN. 
		// Shutter within open to open resolver pos ??
		// Verification of open shutter switches for Heimdal, T-Rex and Magic.
		// Motor power on, brake off. Scientists ask permission - ctrl room executes.
		// To do: LS verification and fault handling.
		(*
		actPower();
		actOpenToOpen();
		//fbOpenToOpen(bAxisDelayPower:=bAxisDelayPower, bAxisDelayDone:=bAxisDelayDone);

		IF bAxesDone AND bDelayOpenToOpen THEN // bDelayOpenToOpen prevents early exit from this state
			//ABS(GVL.astAxes[MAIN.hmiAxisSelection].stStatus.fActPosition - 
			//	aLightShutters[MAIN.hmiAxisSelection].pos[aLightShutters[MAIN.hmiAxisSelection].curPosNbr]) < 1 THEN
			aOpenToOpen[1] := FALSE; // change to aOpenToOpen
			aOpenToOpen[2] := FALSE;
			//actPower();
			eLightShutterSystemState := E_LightShutterSystemStates.Open;
		END_IF
		*)

	// Remove?
	E_LightShutterSystemStates.Adjusting: // Alt: Remove substate and have as option in Open instead
		// Verification of open shutter, switch in question.
		// Switch cams open position +- 2 mm. Motor power on, brake off.
		// To do: LS verification and fault handling.

		(*
		IF GVL.astAxes[MAIN.hmiAxisSelection].stStatus.bEnabled THEN
			GVL.astAxes[MAIN.hmiAxisSelection].stControl.eCommand :=E_MotionFunctions.eJog;
		
			GVL.astAxes[MAIN.hmiAxisSelection].stControl.bJogBwd := bJogB AND 
				GVL.astAxes[MAIN.hmiAxisSelection].stStatus.fActPosition >= 
					GVL_APP.aLightShutters[MAIN.hmiAxisSelection].pos[GVL_APP.aLightShutters[MAIN.hmiAxisSelection].curPosNbr]*0.92; 

			GVL.astAxes[MAIN.hmiAxisSelection].stControl.bJogFwd := bJogF AND 
				GVL.astAxes[MAIN.hmiAxisSelection].stStatus.fActPosition <= 
					GVL_APP.aLightShutters[MAIN.hmiAxisSelection].pos[GVL_APP.aLightShutters[MAIN.hmiAxisSelection].curPosNbr]*1.08;
		END_IF

		IF NOT bJogB AND NOT bJogF THEN
			eLightShutterSystemState := E_LightShutterSystemStates.Open;
		END_IF
		*)

	// Remove?
	E_LightShutterSystemStates.ResetZero:
		// Reset of resolver, top shutter pos against mechanical stop.
		// Motor power on, brake off.
		// To do: Implement sequence: ramp, torque. Fault handling.
		// Should we also record position of Closed shutter?

		(*
		FOR i:=1 TO GVL_APP.nAXIS_NUM DO
			IF aResetZero[i] THEN
				aFbResetZero[i](bResetZero := aResetZero[i], bAxisDelayDone := bAxisDelayDone, axisNbr := i);
			END_IF

		END_FOR

		//fbResetZero(bResetZero := bResetZero, bAxisDelayDone := bAxisDelayDone);

		IF bAxesDone AND NOT bResetZero THEN // ALSO IF NOT PRESSED ANYMORE?
		//IF NOT bResetZero THEN // Transitioning from state - need to check axis status? 
			eLightShutterSystemState := E_LightShutterSystemStates.Open;
		END_IF*)

	E_LightShutterSystemStates.Closing:
		// Resolver monitoring of shutter positions.
		// LSS monitor time for event to happen. Motor power on, brake off
		// To do: Fault handling.

		bEnablePower := TRUE;
		actCascadePower();
		actCascadeClosing();

		IF bAxesDone AND bClosedShutters THEN
			// This one is not safe to check OR bAllDisabled
			eLightShutterSystemState := E_LightShutterSystemStates.ClosedStandby;
		END_IF

	// Remove?
	E_LightShutterSystemStates.Maintenance:
		// Verification of all shutters closed. Motor power off, brake on.
		// As CLOSED OFF, but also administrative permission for port maintenance.

		// Disable alarm from our own switches. But still indicate if 
		// something is open / closed...

		GVL.astAxes[1].stControl.bEnable := FALSE;
		GVL.astAxes[2].stControl.bEnable := FALSE;

		IF bMaintenancePermission THEN
			eLightShutterSystemState := E_LightShutterSystemStates.SinglePortMaintenance_ClosedStandby;
		END_IF


	E_LightShutterSystemStates.SinglePortMaintenance_ClosedStandby:

		GVL.astAxes[1].stControl.bEnable := FALSE; // Do motors really need to be energised here?
		GVL.astAxes[2].stControl.bEnable := FALSE;

		IF bMaintenancePermission THEN
			eLightShutterSystemState := E_LightShutterSystemStates.SinglePortMaintenance_Opening;
		END_IF

		IF bMaintencancePerformed THEN
			eLightShutterSystemState := E_LightShutterSystemStates.Maintenance;
		END_IF


	E_LightShutterSystemStates.SinglePortMaintenance_Opening:
		// Single shutter opening during maintenance of shutter.
		// Local control? Manual jogging? 

		GVL.astAxes[1].stControl.bEnable := TRUE;
		GVL.astAxes[2].stControl.bEnable := TRUE;
		//actMaintenanceOpening();

		IF bAxesDone AND bInPos THEN
			eLightShutterSystemState := E_LightShutterSystemStates.SinglePortMaintenance_Open;
		END_IF


	E_LightShutterSystemStates.SinglePortMaintenance_Open:
		// Single shutter open during maintenance of shutter.
		// Local control?

		GVL.astAxes[MAIN.hmiAxisSelection].stControl.bEnable := FALSE;


	E_LightShutterSystemStates.SinglePortMaintenance_Closing:
		// Single shutter closing during maintenance of shutter.
		// Local control?

		GVL.astAxes[MAIN.hmiAxisSelection].stControl.bEnable := FALSE;


	E_LightShutterSystemStates.LSS_Maintenance:
		GVL.astAxes[MAIN.hmiAxisSelection].stControl.bEnable := FALSE;


	E_LightShutterSystemStates.Fault:
		// Any LSS state machine fault. Two levels of severity: A and B.

		GVL.astAxes[MAIN.hmiAxisSelection].stControl.bEnable := FALSE;

END_CASE

ACTION actCascadeClosing:
// Closes all beamlines, in the future in a cascade to limit power peak.
// To fix: Cascading

FOR i := 1 TO nAXIS_NUM DO

	IF GVL.astAxes[i].stStatus.bEnabled THEN
		GVL.astAxes[i].stControl.eCommand:=E_MotionFunctions.eJog;
		GVL.astAxes[i].stControl.bJogBwd:= GVL.astAxes[i].stStatus.bBwEnabled;	
	END_IF

END_FOR
END_ACTION

ACTION actCascadeHoming:
// Homes all beamlines, in the future in a cascade
// To fix: Cascading

FOR i := 1 TO nAXIS_NUM DO
	IF GVL.astAxes[i].stStatus.bEnabled THEN
		GVL.astAxes[i].stConfig.eHomeSeq := E_HomingRoutines.eHomeToLimit_Bwd;
		GVL.astAxes[i].stControl.eCommand := E_MotionFunctions.eHome;
		GVL.astAxes[i].stControl.bExecute := TRUE;
	END_IF
END_FOR
END_ACTION

ACTION actCascadeOpening:
// Opens all beamlines to the first focal point position, in the future in a cascade
// To do: Cascading

FOR i := 1 TO nAXIS_NUM DO
	IF GVL.astAxes[i].stStatus.fActPosition <> 100 THEN // Change to something sensible
		IF GVL.astAxes[i].stStatus.bEnabled THEN
			GVL.astAxes[i].stControl.fPosition := GVL_APP.aLightShutters[i].pos[1];
			GVL.astAxes[i].stControl.eCommand := E_MotionFunctions.eMoveAbsolute;
			GVL.astAxes[i].stControl.bExecute := TRUE;
		END_IF
	END_IF
	GVL_APP.aLightShutters[i].curPosNbr:=1;
END_FOR
END_ACTION

ACTION actCascadePower:
// Enable power to all beamlines if not disabled, in the future cascading.
// To fix: cascading.

FOR i := 1 TO nAXIS_NUM DO
	GVL.astAxes[i].stControl.bEnable := (bEnablePower AND NOT aDisabled[i]); //OR XOR ar_bPower[i];
END_FOR
END_ACTION

ACTION actDelayDisable:
// Delays the disabeling of each axis

FOR i := 1 TO nAXIS_NUM DO
    aTOF_delayDisable[i](IN:=aJogB[i] OR aJogF[i] OR aResetZero[i] OR aOpenToOpen[i], PT:=T#10S);
END_FOR
END_ACTION

ACTION actDelayDone:
// Delays the bDone of each axis

FOR i := 1 TO nAXIS_NUM DO
    aTON_delayDone[i](IN:=GVL.astAxes[i].stStatus.bDone, PT:=T#1S);
END_FOR
END_ACTION

ACTION actDelayOpenToOpen:
// Delays aOpenToOpen[i] for each axis

FOR i := 1 TO nAXIS_NUM DO
    aTON_delayOpenToOpen[i](IN:=aOpenToOpen[i], PT:=T#0.5S);
END_FOR
END_ACTION

ACTION actFaults:
// Checking for faults which could take the statemachine into a fault state

// Actuator velocity: > 110 mm/s - B
// Actuator stroke time out: > 30 s - A
// Motor torque: > 21.5 Nm - B
// Motor DC Voltage downwards movement: > 850 V - B
// Motor DC Voltage upwards movement: > 600 V - B
// Motor DC Power upwards movement: > 380 W - B
// Applied hold brake position indication: Any feedback signal deviating from what is expected - B
// Resolver position compared with Closed Shutter Indications: Deviation 0.5 mm - A
// Deviation: Resolver position compared with Open Shutter LO: Deviation 2.2 mm (adjustment range +-2 mm) - A
// Deviation: Resolver position compared with Open Shutter HI: Deviation 2.2 mm (adjustment range +-2 mm) - A
// Motor temperature: > 50 C - B
// Servo drive temperature: > 50 C - B
// Homing sequence not fulfilled timeout > 30 s - B

// Should a statemachine take care of these cases? eFaults.A/B?
END_ACTION

ACTION actInitAxis:
// Initialization of axes

GVL_APP.aLightShutters[E_Beamline.Miracles].nbrOfPos := 1;
GVL_APP.aLightShutters[E_Beamline.Heimdal].nbrOfPos := 2;
END_ACTION

ACTION actJog:
// Moves all chosen beamlines

FOR i := 1 TO nAXIS_NUM DO

		IF GVL.astAxes[i].stStatus.bEnabled AND NOT aResetZero[i] AND NOT aOpenToOpen[i] AND NOT aDisabled[i] THEN
			IF (aJogB[i] OR aJogF[i]) THEN
				GVL.astAxes[i].stControl.eCommand :=E_MotionFunctions.eJog;
			END_IF
			
			GVL.astAxes[i].stControl.bJogBwd := aJogB[i] AND 
				GVL.astAxes[i].stStatus.fActPosition >= 
					GVL_APP.aLightShutters[i].pos[GVL_APP.aLightShutters[i].curPosNbr]*0.94; 
		
			GVL.astAxes[i].stControl.bJogFwd := aJogF[i] AND 
				GVL.astAxes[i].stStatus.fActPosition <= 
					GVL_APP.aLightShutters[i].pos[GVL_APP.aLightShutters[i].curPosNbr]*1.06;
		END_IF
		
END_FOR
END_ACTION

ACTION actOpenToOpen:
// Moves all chosen beamlines to chosen position

FOR i := 1 TO nAXIS_NUM DO
	
	IF aOpenToOpen[i] AND NOT aDisabled[i] THEN
		GVL.astAxes[i].stControl.bEnable := TRUE;
		IF GVL.astAxes[i].stStatus.bEnabled THEN
			GVL.astAxes[i].stControl.fPosition := 
				GVL_APP.aLightShutters[i].pos[GVL_APP.aLightShutters[i].curPosNbr];
			GVL.astAxes[i].stControl.eCommand := E_MotionFunctions.eMoveAbsolute;
			GVL.astAxes[i].stControl.bExecute := TRUE;
		END_IF
		
		IF GVL.astAxes[i].stStatus.bDone AND aTON_delayOpenToOpen[i].Q THEN
			aOpenToOpen[i] := FALSE;
		END_IF
		
	ELSIF aDisabled[i] THEN
		aOpenToOpen[i] := FALSE;
	END_IF
	
END_FOR
END_ACTION

ACTION actPositionSwitches:
// Update the array of switches

FOR i := 1 TO nAXIS_NUM DO
	
	GVL_APP.aPosSwitch[i,1] := GVL.astAxes[i].stInputs.bHomeSensor; // Needs change to correct BOOL
	
	IF GVL_APP.aLightShutters[i].nbrOfPos = 2 THEN
		GVL_APP.aPosSwitch[i,2] := bOpenHiFake;
	END_IF
	
END_FOR
END_ACTION

ACTION actPower:
// Enable power to individual beamlines if not disabled.

FOR i := 1 TO nAXIS_NUM DO
	
	IF GVL.astAxes[i].stStatus.bDone THEN
		GVL.astAxes[i].stControl.bEnable := ((aJogB[i] OR aJogF[i] OR aTOF_delayDisable[i].Q OR aOpenToOpen[i] OR aResetZero[i]) AND NOT aDisabled[i]); //OR XOR ar_bPower[i];
	END_IF
	
END_FOR
END_ACTION

ACTION actResetZero:
// Calls a FB_ResetZero for each axis where aResetZero[i] is TRUE

FOR i:=1 TO nAXIS_NUM DO
	
	IF aResetZero[i] AND NOT aDisabled[i] THEN
        aFbResetZero[i](bResetZero := aResetZero[i], bAxisDone:=GVL.astAxes[i].stStatus.bDone, axisNbr := i);
	ELSIF aDisabled[i] THEN
		aResetZero[i] := FALSE;
	END_IF
	
END_FOR
END_ACTION

ACTION actRunMethods:
// Runs methods

//checkAxesEnabled(bOutput => bAxesEnabled);

checkVirtualHomed(bOutput => bAxesHomed);
checkAxesDone(bOutput => bAxesDone);
checkPos(bOutput => bInPos);
checkClosedLimitSwitches(bOutput => bClosedShutters);
checkAllDisabled(bOutput => bAllDisabled);
// checkOpenToOpen(bOutput => bOpenToOpen);
// checkResetZero(bOutput => bResetZero);
// checkJog(bOutput => bJog);
// checkEnabled(bOutput => bAxesEnabled);


//checkAllAxisErrors(bOutput => bAxisErrorsPresent);
//checkErrorState(bOutput => bFunctionInErrorState);*)
END_ACTION

ACTION actSavePos:
// Saves the current position of all axes to aLightShutters. NOT USED

FOR i := 1 TO nAXIS_NUM DO
	GVL_APP.aLightShutters[i].pos[GVL_APP.aLightShutters[MAIN.hmiAxisSelection].curPosNbr] := GVL.astAxes[i].stStatus.fActPosition;
END_FOR
END_ACTION

(*Method to check if all axes are disabled.
Only returns TRUE if all axes are enabled.*)
METHOD checkAllDisabled: BOOL
VAR_OUTPUT
    bOutput: BOOL := TRUE;
END_VAR

VAR
	i : DINT := 1;
END_VAR
FOR i := 1 TO nAXIS_NUM DO
	IF NOT aDisabled[i] THEN
		bOutput := FALSE;
		EXIT;
	END_IF
END_FOR
END_METHOD

(*Method to check if all axes are Done.
Only returns TRUE if all axes are Done*)
METHOD checkAxesDone: BOOL
VAR_OUTPUT
    bOutput: BOOL := TRUE;
END_VAR

VAR
	i : DINT := 1;
END_VAR
FOR i := 1 TO nAXIS_NUM DO
	IF NOT aDisabled[i] THEN
		IF NOT GVL.astAxes[i].stStatus.bDone THEN
    		bOutput := FALSE;
			EXIT;
		END_IF
	END_IF
END_FOR
END_METHOD

(*Method to check if all axes are closed. Ignores a axis if it is disabled.
Only returns TRUE if all axes are closed*)
METHOD checkClosedLimitSwitches: BOOL
VAR_OUTPUT
    bOutput: BOOL := TRUE;
END_VAR

VAR
	i : DINT := 1;
END_VAR
// Needs fix, dealing with e.g. fPos 0.

FOR i := 1 TO nAXIS_NUM DO
	IF GVL.astAxes[i].stInputs.bLimitBwd AND NOT aDisabled[i] THEN
		bOutput := FALSE;
		EXIT;
	END_IF
END_FOR
END_METHOD

(*Method to check if the axes are homed/the calibration flag is present.
Only returns TRUE if all axes are homed *)
METHOD checkEnabled: BOOL
VAR_OUTPUT
    bOutput: BOOL:= FALSE;
END_VAR

VAR
	i : DINT := 1;
END_VAR
FOR i := 1 TO nAXIS_NUM DO
	IF GVL.astAxes[i].stStatus.bEnabled THEN
    	bOutput := TRUE;
		EXIT;
	END_IF
END_FOR
END_METHOD

(*Method to check if all axes are disabled.
Only returns TRUE if all axes are enabled.*)
METHOD checkJog: BOOL
VAR_OUTPUT
    bOutput: BOOL := FALSE;
END_VAR

VAR
	i : DINT := 1;
END_VAR
FOR i := 1 TO nAXIS_NUM DO
	IF aJogB[i] OR aJogF[i] THEN
		bOutput := TRUE;
		EXIT;
	END_IF
END_FOR
END_METHOD

(*Method to check if all axes are disabled.
Only returns TRUE if all axes are enabled.*)
METHOD checkOpenToOpen: BOOL
VAR_OUTPUT
    bOutput: BOOL := FALSE;
END_VAR

VAR
	i : DINT := 1;
END_VAR
FOR i := 1 TO nAXIS_NUM DO
	IF aOpenToOpen[i] THEN
		bOutput := TRUE;
		EXIT;
	END_IF
END_FOR
END_METHOD

(*Method to check if all axes are withing 10 % of its set value.
Only returns TRUE if all axes are within 10% of fPosition.*)
METHOD checkPos: BOOL
VAR_OUTPUT
    bOutput: BOOL := TRUE;
END_VAR

VAR
	i : DINT := 1;
END_VAR
// Needs fix, dealing with e.g. fPos 0.

FOR i := 1 TO nAXIS_NUM DO
	IF NOT aDisabled[i] THEN // Check if beamline is disabled/enabled
		IF GVL.astAxes[i].stStatus.fActPosition < GVL.astAxes[i].stControl.fPosition*0.9 
		OR GVL.astAxes[i].stStatus.fActPosition > GVL.astAxes[i].stControl.fPosition*1.10 THEN  // Add something about position?
    		bOutput := FALSE;
			EXIT;
		END_IF
	END_IF
END_FOR
END_METHOD

(*Method to check if all axes are disabled.
Only returns TRUE if all axes are enabled.*)
METHOD checkResetZero: BOOL
VAR_OUTPUT
    bOutput: BOOL := FALSE;
END_VAR

VAR
	i : DINT := 1;
END_VAR
FOR i := 1 TO nAXIS_NUM DO
	IF aResetZero[i] THEN
		bOutput := TRUE;
		EXIT;
	END_IF
END_FOR
END_METHOD

(*Method to check if the axes are homed/the calibration flag is present.
Only returns TRUE if all axes are homed *)
METHOD checkVirtualHomed: BOOL
VAR_OUTPUT
    bOutput: BOOL:= TRUE;
END_VAR

VAR
	i : DINT := 1;
END_VAR
FOR i := 1 TO nAXIS_NUM DO
	IF NOT GVL.astAxes[i].stStatus.bHomed THEN
    	bOutput := FALSE;
		EXIT;
	END_IF
END_FOR
END_METHOD

END_PROGRAM

// ---- POUs/Application_Specific/Applications/SeqRangePos.TcPOU
PROGRAM SeqRangePos
VAR
//Define all necessary variables for your application
	bManual: BOOL := FALSE;
	//bResult: BOOL := FALSE;
	eMotorState: E_SeqRangePosStates := E_SeqRangePosStates.INIT;
	
	bAxesEnabled: BOOL := FALSE; // Should be a word instead?
	bEnable: BOOL;
	bMotorsHomed: BOOL;
	bHoming: BOOL;
	//bPos1: BOOL := FALSE;
	//bPos2: BOOL := FALSE;
	//bPos0: BOOL := TRUE;
	bJogB: BOOL := FALSE;
	bJogF: BOOL := FALSE;
	bAdjust: BOOL := FALSE;
	dPos: DWORD;
	dPos_old: DWORD;

END_VAR

actRunMethods();
IF bManual THEN
	dPos.1 := 1;
//ELSIF NOT bManual THEN
	//dPos.1 := 0;
END_IF

IF dPos <> 0 AND dPos <> dPos_old THEN
	dPos := dPos_old XOR dPos;
	dPos_old := dPos;
ELSIF dPos = 0 THEN
	dPos_old := dPos;
END_IF


CASE eMotorState OF
	E_SeqRangePosStates.INIT:
		IF bAxesEnabled AND bEnable THEN
			eMotorState := E_SeqRangePosStates.CHECK_HOME_STATUS;
		END_IF
	
	E_SeqRangePosStates.CHECK_HOME_STATUS:
		IF bMotorsHomed THEN
			eMotorState := E_SeqRangePosStates.CHECK_HOME_COMPLETE;
			bHoming := FALSE;
		END_IF
		
		GVL.astAxes[1].stConfig.eHomeSeq := E_HomingRoutines.eHomeToLimit_Bwd;
		GVL.astAxes[1].stControl.eCommand := E_MotionFunctions.eHome;
		GVL.astAxes[1].stControl.bExecute := TRUE;
		eMotorState := E_SeqRangePosStates.CHECK_HOME_COMPLETE;
		
	E_SeqRangePosStates.CHECK_HOME_COMPLETE:
		IF bMotorsHomed THEN
			eMotorState := E_SeqRangePosStates.MOTOR_OPERATIONAL;
		END_IF
		
	E_SeqRangePosStates.MOTOR_OPERATIONAL:
		IF dPos.0 THEN
			IF GVL.astAxes[1].stControl.fPosition <> 10 AND GVL.astAxes[1].stStatus.fActPosition <> 10 THEN
				GVL.astAxes[1].stControl.fPosition:=10;
				GVL.astAxes[MAIN.hmiAxisSelection].stControl.eCommand:=E_MotionFunctions.eMoveAbsolute;
				GVL.astAxes[MAIN.hmiAxisSelection].stControl.bExecute:=TRUE;
			END_IF
			
			IF GVL.astAxes[1].stStatus.bDone THEN
				eMotorState := E_SeqRangePosStates.POS_ZERO;
			END_IF
		
		ELSIF dPos.1 THEN
			IF GVL.astAxes[1].stControl.fPosition <> 100 AND NOT bAdjust THEN
				GVL.astAxes[1].stControl.fPosition:=100;
				GVL.astAxes[MAIN.hmiAxisSelection].stControl.eCommand:=E_MotionFunctions.eMoveAbsolute;
				GVL.astAxes[MAIN.hmiAxisSelection].stControl.bExecute:=TRUE;	
			ELSIF bAdjust THEN
				GVL.astAxes[1].stControl.eCommand :=E_MotionFunctions.eJog;
				GVL.astAxes[1].stControl.bJogBwd := bJogB AND GVL.astAxes[1].stStatus.fActPosition >= 90;
				GVL.astAxes[1].stControl.bJogFwd := bJogF AND GVL.astAxes[1].stStatus.fActPosition <= 110;
			END_IF
			
			
			//eMotorState := E_SeqRangePosStates.POS_ONE;
			
			//IF GVL.astAxes[1].stStatuS.bDone THEN
			//	eMotorState := E_SeqRangePosStates.POS_ONE;
			//END_IF
		(*ELSIF bPOS2 THEN
			//eMotorState := E_SeqRangePosStates.POS_ONE;
			GVL.astAxes[1].stControl.fPosition:=175;
			GVL.astAxes[1].stControl.eCommand:=E_MotionFunctions.eMoveAbsolute;
			GVL.astAxes[1].stControl.bExecute:=TRUE;
			IF GVL.astAxes[1].stStatus.bDone THEN
				eMotorState := E_SeqRangePosStates.POS_ONE;
			END_IF *)
		END_IF
		
	E_SeqRangePosStates.POS_ZERO:
		//Jogging not allowed
		IF GVL.astAxes[1].stStatus.bDone THEN
				eMotorState := E_SeqRangePosStates.MOTOR_OPERATIONAL;
		END_IF
	
	//E_SeqRangePosStates.POSITIONING:
		//Check if moving??
		
	E_SeqRangePosStates.POS_ONE:
		GVL.astAxes[1].stControl.eCommand:=E_MotionFunctions.eJog;
		GVL.astAxes[1].stControl.bJogBwd:= bJogB;
		GVL.astAxes[1].stControl.bJogBwd:= bJogF;
		

	
	//E_SeqRangePosStates.POS_TWO:
		//
END_CASE

ACTION actRunMethods:
checkAxesEnabled(bOutput => bAxesEnabled);
//checkBladesHomed(bOutput => bBladesHomed);
checkVirtualHomed(bOutput => bMotorsHomed);
//checkBladesCoupled(bOutput => bBladesCoupled);
//checkBladesUncoupled(bOutput => bBladesUncoupled);
//checkAllAxisErrors(bOutput => bAxisErrorsPresent);
//checkErrorState(bOutput => bFunctionInErrorState);*)
END_ACTION

(*Method to check if all axes (real and virtual) are enabled.
Only returns TRUE if BOTH blades are homed*)
METHOD checkAxesEnabled: BOOL
VAR_OUTPUT
    bOutput: BOOL:= TRUE;
END_VAR
IF NOT GVL.astAxes[1].stStatus.bEnabled THEN
    bOutput := FALSE;
END_IF
(*IF NOT GVL.astAxes[iBladePositive].stStatus.bEnabled THEN
    bOutput := FALSE;
END_IF
IF NOT GVL.astAxes[iGapSize].stStatus.bEnabled THEN
    bOutput := FALSE;
END_IF
IF NOT GVL.astAxes[iGapCentre].stStatus.bEnabled THEN
    bOutput := FALSE;
END_IF*)
END_METHOD

(*Method to check if the virtual axes for gap size and gap centre are homed/the calibration flag is present.
Only returns TRUE if BOTH virtual axes are homed *)
METHOD checkVirtualHomed: BOOL
VAR_OUTPUT
    bOutput: BOOL:= TRUE;
END_VAR
IF NOT GVL.astAxes[1].stStatus.bHomed THEN
    bOutput := FALSE;
END_IF
//IF NOT GVL.astAxes[1].stStatus.bHomed THEN
//    bOutput := FALSE;
////END_IF
END_METHOD

END_PROGRAM

// ---- tc_pils/tc_pils_app_specific/POUs/PILS_DEVICES.TcPOU
PROGRAM PILS_DEVICES
VAR
END_VAR

//Interface between PILS and AXIS
//Example code of how to link the axis and PILS
fbMotorM1(stAxisStruct:= astAxes[1], stDeviceStructPILS:= stMotorM1, stAxisPar:= stMotorM1Param);
fbMotorM2(stAxisStruct:= astAxes[2], stDeviceStructPILS:= stMotorM2, stAxisPar:= stMotorM2Param);
stPowerSwitchesAxis1.nValue:= BOOL_TO_INT(Axis_Template.bPowerSwitchesAxis1);
stPowerSwitchesAxis2.nValue:= BOOL_TO_INT(Axis_Template.bPowerSwitchesAxis2);
//stPowerSwitchesAxis1Ctr.nCurrentValue:= BOOL_TO_INT(Axis_Template.bPowerSwitchesAxis1);
//stPowerSwitchesAxis1Ctr.nTargetValue:= BOOL_TO_INT(Axis_Template.bPowerSwitchesAxis1);

//stMotor1Temp.fValue := Axis_1.fMotTemp1;
//stMotorM1EncoderRaw.nValue := nEncoderValueAxis1;

END_PROGRAM

// ---- GlobalTextList.TcGTLO
TEXTLIST GlobalTextList
  947 = '   LocalMode'
  972 = '  bLocalMode'
  587 = '%1d'
  951 = '%2.2f'
  543 = '%2.4f'
  982 = '%d'
  235 = '%f'
  39 = '%n'
  821 = '%s'
  916 = '%time_t'
  940 = '%x'
  1835 = '1'
  626 = '2'
  952 = 'actPos'
  953 = 'actVel'
  5 = 'Add closed switches \nfrom us and PSS'
  365 = 'Add closed switches \nfrom us and PSS\n\nAdd incremental choice'
  1153 = 'Add closed switches from us and PSS'
  29 = 'Adjusting'
  110 = 'AXESMAX'
  256 = 'Axis'
  1718 = 'Axis Error'
  425 = 'axisSe'
  107 = 'axisSel'
  250 = 'bAdjusting'
  945 = 'bBusy'
  950 = 'bBwEnabled'
  220 = 'bClosing'
  633 = 'bCoammandAborted'
  225 = 'bCommandAborted'
  946 = 'bDone'
  943 = 'bEnabled'
  941 = 'bError'
  102 = 'bExecute'
  999 = 'bExtended'
  949 = 'bFwEnabled'
  297 = 'bGeared'
  1303 = 'bHome'
  948 = 'bHomed'
  944 = 'bCommandAborted'
  183 = 'bInterlock'
  382 = 'bJog'
  498 = 'bJogB'
  400 = 'bJogF'
  544 = 'bLSS_On'
  128 = 'bLSSOpen'
  485 = 'bMovingExtend'
  648 = 'bMovingExtract'
  998 = 'bMovingRetract'
  1300 = 'bOpenToOpen'
  511 = 'bPermit'
  450 = 'bPoweEncAxis1'
  40 = 'bPoweEncAxis2'
  886 = 'bPowerSwitches1'
  87 = 'bPowerSwitchesAxis1'
  161 = 'bPowerSwitchesAxis2'
  963 = 'bPSSPermit'
  352 = 'bReset'
  226 = 'bRetracted'
  933 = 'bValveOn'
  786 = 'Bwd Enable'
  634 = 'Closed'
  119 = 'Closed\nLSS / PSS'
  62 = 'Closed LSS - PSS - PSS'
  159 = 'Closed LSS / PSS'
  907 = 'Closed Off'
  1624 = 'Closed Shutter'
  1955 = 'Closed Shutter - LSS - PSS - PSS'
  1735 = 'Closed Shutter LSS / PSS'
  1806 = 'Closed Shutters'
  1206 = 'Closed Standby'
  1186 = 'ClosedOff'
  646 = 'ClosedStandby'
  1385 = 'Closing'
  908 = 'Confirmed Ready'
  402 = 'ConfirmedReady'
  503 = 'Cooling Down'
  1214 = 'CoolingDown'
  602 = 'Disable'
  1630 = 'Disable Beamline Operation'
  986 = 'ehomeDirect'
  350 = 'eHomeDirect'
  180 = 'eHomeEncPulseBwd'
  198 = 'eHomeToEncPulse_Bwd'
  510 = 'eHomeToEncPulse_Fwd'
  287 = 'eHomeToEncPulse_viaBwdLimit'
  683 = 'eHomeToEncPulse_viaFwdLimit'
  312 = 'eHomeToLimit_Bwd'
  635 = 'eHomeToLimit_Fwd'
  150 = 'eHomeToRef_Bwd'
  861 = 'eHomeToRef_Fwd'
  2127 = 'eHomeTorque'
  311 = 'eHomeTorque - Back'
  1094 = 'eHomeTorque - Fwd'
  313 = 'Elapsed time'
  104 = 'ENABLE'
  1158 = 'Enable'
  1879 = 'Enable / Disable Operation'
  106 = 'ENABLE BW'
  105 = 'ENABLE FW'
  961 = 'Enable/Disable Operation'
  109 = 'English'
  1004 = 'eReadParameter'
  939 = 'errID'
  768 = 'eWriteParameter'
  768 = 'eWriteParameter'
  937 = 'E_PneumaticErrors'
  333 = 'E_PneumaticMode'
  463 = 'E_PneumaticMode Selection'
  962 = 'f'
  1422 = 'fAccel'
  955 = 'fAcceleration'
  324 = 'fDecel'
  956 = 'fDeceleration'
  531 = 'fHomeFinishDistance'
  613 = 'fHomePosition'
  157 = 'fHomePositions'
  957 = 'fPosition'
  149 = 'fRatio'
  781 = 'fReadAxisParameter'
  954 = 'fVelocity'
  668 = 'Fwd Enable'
  688 = 'fWriteAxisParameter'
  299 = 'gearIn'
  717 = 'gearInMultiMaster'
  300 = 'gearOut'
  523 = 'halt'
  282 = 'Heimdal'
  1126 = 'HEIMDAL'
  1306 = 'Hide this and think\nabout how it is to'
  837 = 'Hide this and think\nabout how it is to\nbe accessed'
  123 = 'HOME'
  568 = 'Home'
  169 = 'homeDirect'
  917 = 'HomeDirect'
  175 = 'HomeEncBwd'
  411 = 'HomeEncBwdLim'
  723 = 'HomeEncFwd'
  777 = 'HomeEncFwdLim'
  547 = 'HomeEncPulBwdLim'
  1453 = 'HomeEncPulseBwd'
  1440 = 'HomeEnc_BwdLim'
  820 = 'HomeEnc_BwdLimit'
  906 = 'HomeLimBwd'
  909 = 'HomeLimFwd'
  1028 = 'HomeRefBwd'
  996 = 'HomeRefFwd'
  566 = 'homeSensorNeg'
  677 = 'homeSensorPos'
  263 = 'HomeToRefBwd'
  1223 = 'INIT'
  784 = 'Interlock Bwd'
  505 = 'Interlock Fwd'
  1504 = 'Jog Down'
  339 = 'Jog Up'
  831 = 'Jog Up / Down'
  385 = 'Jog Up/Down'
  116 = 'jogBw'
  117 = 'jogFw'
  19 = 'Limit switches simulation'
  919 = 'LimitBwd'
  459 = 'LimitFwd'
  870 = 'Local Mode'
  1529 = 'LOKI'
  2035 = 'LSS'
  651 = 'LSS Open'
  682 = 'LSS Stateas'
  1030 = 'LSS States'
  1052 = 'Maintenance'
  205 = 'Manual Control'
  298 = 'masterGear'
  328 = 'MIRACLES'
  460 = 'Mode Selection'
  118 = 'Mode selection'
  111 = 'moveAbsolute'
  114 = 'moveModulo'
  113 = 'moveRelative'
  112 = 'moveVelocity'
  841 = 'Neutron Factory States'
  575 = 'nIndex'
  496 = 'Not Confirmed Ready'
  130 = 'NotConfirmedReady'
  716 = 'nTimeToExtend'
  787 = 'nTimeToExtend(ms)'
  992 = 'nTimeToExtend(s)'
  929 = 'nTimeToRetract'
  444 = 'nTimeToRetract(ms)'
  995 = 'nTimeToRetract(s)'
  960 = 'Open'
  1324 = 'OPEN - HI'
  1127 = 'OPEN - LO'
  774 = 'Open To Open'
  214 = 'Opening'
  1183 = 'OpenToOpen'
  330 = 'Pneumatic Axis Selection'
  958 = 'Pneumatic AxisSelection'
  694 = 'Pneumatics'
  652 = 'Pos OPEN - LO'
  1197 = 'Position OPEN - LO'
  1423 = 'PSS'
  1516 = 'PSS Permission'
  1182 = 'PSS Permission\n\nServo Drive Powered'
  92 = 'PSS Permission\n\nServo Drives\nPowered'
  850 = 'PSS Permission\n\nServo Drives Powered'
  1174 = 'PSS Permit'
  184 = 'PSS Power'
  942 = 'reset'
  1022 = 'Reset'
  807 = 'Reset Error'
  1248 = 'Reset To Zero'
  858 = 'Reset Zero'
  1522 = 'Servo \nMotor'
  611 = 'shomeDirect'
  227 = 'Single Solenoid Manual'
  761 = 'Single Solenoid PLC'
  581 = 'Single Solenoid PLC ON'
  959 = 'Sngle solenoid PLC'
  466 = 'Sngle solenoid PLC '
  855 = 'sStatus'
  211 = 'Start Extend'
  259 = 'Start Retract'
  410 = 'Start Up'
  1073 = 'StartUp'
  889 = 'Stepper \nMotor'
  822 = 'Stepper Motor'
  115 = 'stop'
  1658 = 'Test'
  108 = 'Test Language'
  730 = 'To do:'
  1036 = 'To do:\n* Transitions when aborting'
  1232 = 'To do:\n*Transitions when aborting\n*Fault state'
  433 = 'To do:\n*Transitions when aborting\n*Fault state\n*Substate as fb:s?'
  1048 = 'To do:\n*Transitions when aborting\n*Fault state\n*Torque'
  731 = 'To do:\n*Transitions when aborting\n*Fault state\n*Torque Homing'
  2163 = 'To do:\n*Transitions when aborting\n*RTrig for first entry in state'
  2038 = 'To do:\n*Transitions when aborting\n*RTrig for first entry in state\n*Fault state'
  1997 = 'To do:\n*Transitions when aborting\n*RTrig for first entry in state\n*Fault state\n*Substate as fb:s?'
  66 = 'To do:\n*Transitions when aborting\n*RTrig for first entry in state?'
  103 = 'toggle'
  1313 = 'Up'
  445 = 'Write'
  322 = 'WriteParameters'
END_TEXTLIST

// ---- VISUs/AcceleratorStates.TcVIS
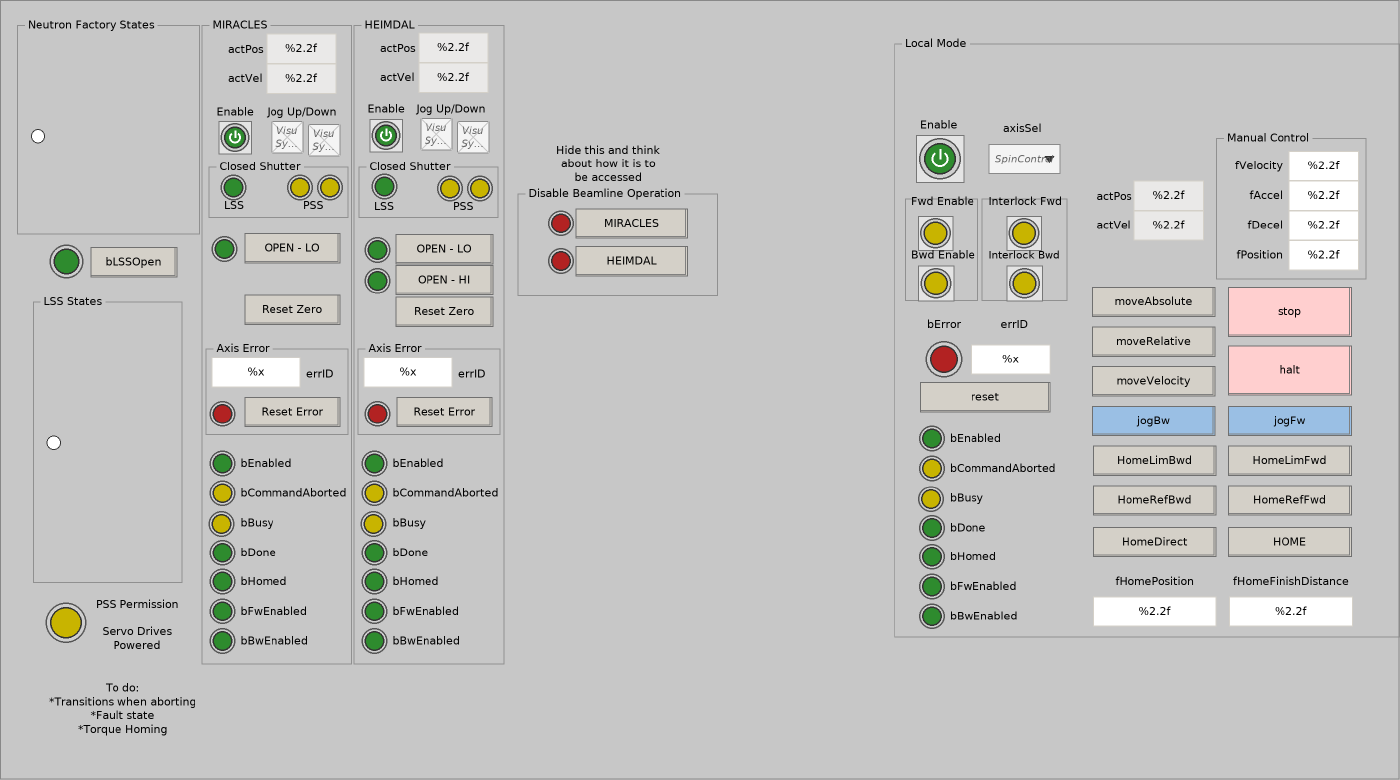
VISUALIZATION AcceleratorStates  // 1409x786
    GroupBox (361,160 140x59), "Closed Shutter"
    GroupBox (210,160 140x59), "Closed Shutter"
    GroupBox (203,17 151x652), "MIRACLES"
        Textfield (11,18 54x30), "actPos", text list: 'languageTable', text index: "actposition"
        Textfield (65,17 70x30), "%2.2f", text variable: GVL.astAxes[1].stStatus.fActPosition
        Textfield (15,47 49x30), "actVel", text list: 'languageTable', text index: "actVelocity"
        Textfield (65,47 70x30), "%2.2f", text variable: GVL.astAxes[1].stStatus.fActVelocity
        Lamp1 (6,385 30x30), variable: GVL.astAxes[1].stStatus.bError, style: Lamp-Lamp1-Red
        PowerSwitch (16,105 35x33), variable: GVL.astAxes[1].stControl.bEnable, behaviour: TOGGLE, style: Switch-PowerSwitch-Green
        Lamp1 (8,219 30x30), variable: GVL.astAxes[1].stInputs.bHomeSensor, style: Lamp-Lamp1-Green
        Button (43,218 96x30), "OPEN - LO", pressed state: LightShutterSystemStates.aOpenToOpen[1]
            toggle LightShutterSystemStates.aOpenToOpen[1]
            OnMouseDown: execute {
                //MAIN.hmiAxisSelection := 1;
                GVL_APP.aLightShutters[1].curPosNbr:=1;
            }
        Button (43,383 96x30), "Reset Error", pressed state: GVL.astAxes[1].stControl.bReset, text list: 'languageTable', text index: "reset"
            OnMouseClick: toggle GVL.astAxes[1].stControl.bReset
        Image (70,105 32x32), image: VisuSymbols.Symbols.ArrowBoldUp
            OnMouseUp: execute { LightShutterSystemStates.aJogF[1] := FALSE; }
            OnMouseDown: execute { LightShutterSystemStates.aJogF[1] := TRUE; }
        Image (107,108 32x32), image: VisuSymbols.Symbols.ArrowBoldDown
            OnMouseDown: execute { LightShutterSystemStates.aJogB[1] := TRUE; }
            OnMouseUp: execute { LightShutterSystemStates.aJogB[1] := FALSE; }
        Textfield (12,83 63x26), "Enable", text list: 'languageTable', text index: "enable"
        Textfield (63,83 82x26), "Jog Up/Down", text list: 'languageTable', text index: "jogUpDown"
        Lamp1 (17,157 30x30), variable: NOT(GVL.astAxes[1].stInputs.bLimitBwd), style: Lamp-Lamp1-Green
        Button (43,280 96x30), "Reset Zero"
            toggle LightShutterSystemStates.aResetZero[1]
            OnMouseClick: execute { MAIN.hmiAxisSelection := 1; }
        Textfield (10,343 89x30), "%x", text variable: GVL.astAxes[1].stStatus.nErrorID
        Lamp1 (114,157 30x30), variable: NOT(GVL.astAxes[1].stInputs.bLimitBwd), style: Lamp-Lamp1-Yellow
        Lamp1 (84,157 30x30), variable: NOT(GVL.astAxes[1].stInputs.bLimitBwd), style: Lamp-Lamp1-Yellow
        Label (10,175 45x30), "LSS"
        Label (90,175 45x30), "PSS"
    GroupBox (356,17 151x652), "HEIMDAL"
        Textfield (15,17 50x30), "actPos", text list: "languageSupport", text index: "actposition"
        Textfield (65,24 70x30), "%2.2f", text variable: GVL.astAxes[MAIN.hmiAxisSelection].stStatus.fActPosition
        Button (42,219 98x30), "OPEN - LO", pressed state: LightShutterSystemStates.aOpenToOpen[2]
            toggle LightShutterSystemStates.aOpenToOpen[2]
            OnMouseDown: execute {
                //MAIN.hmiAxisSelection := 2;
                GVL_APP.aLightShutters[2].curPosNbr:=1;
            }
        Lamp1 (9,220 30x30), variable: GVL.astAxes[2].stInputs.bHomeSensor, style: Lamp-Lamp1-Green
        Lamp1 (9,251 30x30), variable: LightShutterSystemStates.bOpenHiFake, style: Lamp-Lamp1-Green
        PowerSwitch (15,103 35x33), variable: GVL.astAxes[2].stControl.bEnable, behaviour: TOGGLE, style: Switch-PowerSwitch-Green
        Textfield (11,80 57x26), "Enable", text list: 'languageTable', text index: "enable"
        Button (42,282 98x30), "Reset Zero"
            toggle LightShutterSystemStates.aResetZero[2]
            OnMouseClick: execute { MAIN.hmiAxisSelection := 2; }
        Textfield (10,343 89x30), "%x", text variable: GVL.astAxes[2].stStatus.nErrorID
        Lamp1 (16,156 30x30), variable: NOT(GVL.astAxes[2].stInputs.bLimitBwd), style: Lamp-Lamp1-Green
    GroupBox (360,343 143x95), "Axis Error"
        Lamp1 (5,59 30x30), variable: GVL.astAxes[2].stStatus.bError, style: Lamp-Lamp1-Red
        Button (39,57 96x30), "Reset Error", pressed state: GVL.astAxes[2].stControl.bReset, text list: 'languageTable', text index: "reset"
            OnMouseClick: toggle GVL.astAxes[2].stControl.bReset
    GroupBox (207,343 143x95), "Axis Error"
    GroupBox (900,36 509x606), "Local Mode"
        Textfield (317,116 77x30), "fVelocity", text list: 'languageTable', text index: "fVelocity"
        Textfield (397,116 70x30), "%2.2f", text variable: GVL.astAxes[MAIN.hmiAxisSelection].stControl.fVelocity
            OnMouseClick: write the text variable via Default
        Textfield (315,146 79x30), "fAccel", text list: 'languageTable', text index: "fAcceleration"
        Textfield (397,146 70x30), "%2.2f", text variable: GVL.astAxes[MAIN.hmiAxisSelection].stControl.fAcceleration
            OnMouseClick: write the text variable via Default
        Textfield (315,176 79x30), "fDecel", text list: 'languageTable', text index: "fDeceleration"
        Textfield (397,176 70x30), "%2.2f", text variable: GVL.astAxes[MAIN.hmiAxisSelection].stControl.fDeceleration
            OnMouseClick: write the text variable via Default
        Textfield (312,206 82x30), "fPosition", text list: 'languageTable', text index: "fPosition"
        Textfield (397,206 70x30), "%2.2f", text variable: GVL.astAxes[MAIN.hmiAxisSelection].stControl.fPosition
            OnMouseClick: write the text variable via Default
        Textfield (241,146 70x30), "%2.2f", text variable: GVL.astAxes[MAIN.hmiAxisSelection].stStatus.fActPosition
        Textfield (193,176 48x30), "actVel", text list: 'languageTable', text index: "actVelocity"
        Textfield (241,176 70x30), "%2.2f", text variable: GVL.astAxes[MAIN.hmiAxisSelection].stStatus.fActVelocity
        Textfield (194,147 48x30), "actPos", text list: 'languageTable', text index: "actposition"
        Textfield (104,276 57x30), "errID", text list: 'languageTable', text index: "errID"
        Textfield (77,311 80x30), "%x", text variable: GVL.astAxes[MAIN.hmiAxisSelection].stStatus.nErrorID
        Lamp1 (28,305 44x42), variable: GVL.astAxes[MAIN.hmiAxisSelection].stStatus.bError, style: Lamp-Lamp1-Red
        Textfield (30,276 79x30), "bError", text list: 'languageTable', text index: "bError"
        Textfield (86,81 86x25), "axisSel", text variable: GVL_APP.nAXIS_NUM, text list: "languageSupport", text index: "axisSel"
    GroupBox (17,17 184x219), "Neutron Factory States"
        RadioButton (12,20 158x200), variable: LightShutterSystemStates.eNeutronFactoryState
            Areas[0]: Text=Disable
            Areas[1]: Text=Maintenance
            Areas[2]: Text=Start Up
            Areas[3]: Text=Cooling Down
            Areas[4]: Text=Not Confirmed Ready
            Areas[5]: Text=Confirmed Ready
    GroupBox (911,192 73x111)
    GroupBox (988,192 86x111)
    PushSwitchLed (924,214 35x42), variable: GVL.astAxes[MAIN.hmiAxisSelection].stInputs.bLimitFwd, behaviour: TOGGLE, style: Switch-PushSwitchLed-Yellow
    PushSwitchLed (924,266 36x39), variable: GVL.astAxes[MAIN.hmiAxisSelection].stInputs.bLimitBwd, behaviour: TOGGLE, style: Switch-PushSwitchLed-Yellow
    SpinControl (995,145 72x30), variable: MAIN.hmiAxisSelection
        p651134158: GVL_APP.nAXIS_NUM
    PushSwitchLed (1013,214 35x42), variable: GVL.astAxes[MAIN.hmiAxisSelection].stControl.bInterlockFwd, behaviour: TOGGLE, style: Switch-PushSwitchLed-Yellow
    PushSwitchLed (1013,266 36x39), variable: GVL.astAxes[MAIN.hmiAxisSelection].stControl.bInterlockBwd, behaviour: TOGGLE, style: Switch-PushSwitchLed-Yellow
    Textfield (914,190 76x26), "Fwd Enable", text list: 'languageSupport', text index: "enFW"
    Textfield (914,244 76x26), "Bwd Enable", text list: 'languageSupport', text index: "enBW"
    Textfield (992,190 76x26), "Interlock Fwd", text list: 'languageSupport', text index: "bAxisInterlockFwd"
    Textfield (992,244 76x26), "Interlock Bwd", text list: 'languageSupport', text index: "bAxisInterlockBwd"
    Lamp1 (923,427 30x30), variable: GVL.astAxes[MAIN.hmiAxisSelection].stStatus.bEnabled, style: Lamp-Lamp1-Green
    Textfield (953,427 117x30), "bEnabled", text list: 'languageTable', text index: "bEnabled"
    Lamp1 (923,457 30x30), variable: GVL.astAxes[MAIN.hmiAxisSelection].stStatus.bCommandAborted, style: Lamp-Lamp1-Yellow
    Textfield (953,457 117x30), "bCommandAborted", text list: 'languageTable', text index: "bWarning"
    Textfield (953,487 117x30), "bBusy", text list: 'languageTable', text index: "bBusy"
    Lamp1 (923,517 30x30), variable: GVL.astAxes[MAIN.hmiAxisSelection].stStatus.bDone, style: Lamp-Lamp1-Green
    Textfield (953,517 117x30), "bDone", text list: 'languageTable', text index: "bDone"
    Lamp1 (923,546 30x30), variable: GVL.astAxes[MAIN.hmiAxisSelection].stStatus.bHomed, style: Lamp-Lamp1-Green
    Textfield (953,546 117x30), "bHomed", text list: 'languageTable', text index: "bHomed"
    Lamp1 (923,576 30x30), variable: GVL.astAxes[MAIN.hmiAxisSelection].stStatus.bFwEnabled AND NOT GVL.astAxes[MAIN.hmiAxisSelection].stStatus.bInterlockedFwd, style: Lamp-Lamp1-Green
    Lamp1 (923,606 30x30), variable: GVL.astAxes[MAIN.hmiAxisSelection].stStatus.bBwEnabled AND NOT GVL.astAxes[MAIN.hmiAxisSelection].stStatus.bInterlockedBwd, style: Lamp-Lamp1-Green
    Textfield (953,576 117x30), "bFwEnabled", text list: 'languageTable', text index: "bFwEnabled"
    Textfield (953,606 117x30), "bBwEnabled", text list: 'languageTable', text index: "bBwEnabled"
    Lamp1 (922,488 30x30), variable: GVL.astAxes[MAIN.hmiAxisSelection].stStatus.bBusy, style: Lamp-Lamp1-Yellow
    Button (1099,289 124x30), "moveAbsolute", text list: 'languageTable', text index: "moveAbsolute"
        OnMouseClick: execute { GVL.astAxes[MAIN.hmiAxisSelection].stControl.eCommand:=E_MotionFunctions.eMoveAbsolute; GVL.astAxes[MAIN.hmiAxisSelection].stControl.bExecute:=TRUE; }
    Button (1099,369 124x30), "moveVelocity", input disabled if: GVL.astAxes[MAIN.hmiAxisSelection].stStatus.bGeared, text list: 'languageTable', text index: "moveVelocity"
        OnMouseClick: execute { GVL.astAxes[Main.hmiAxisSelection].stControl.eCommand:=E_MotionFunctions.eMoveVelocity; GVL.astAxes[Main.hmiAxisSelection].stControl.bExecute:=TRUE; }
    Button (1099,329 124x30), "moveRelative", input disabled if: GVL.astAxes[MAIN.hmiAxisSelection].stStatus.bGeared, text list: 'languageTable', text index: "moveRelative"
        OnMouseClick: execute { GVL.astAxes[Main.hmiAxisSelection].stControl.eCommand:=E_MotionFunctions.eMoveRelative; GVL.astAxes[Main.hmiAxisSelection].stControl.bExecute:=TRUE; }
    Button (1236,289 124x50), "stop", pressed state: GVL.astAxes[Main.hmiAxisSelection].stControl.bStop, input disabled if: GVL.astAxes[MAIN.hmiAxisSelection].stStatus.bGeared, text list: 'languageTable', text index: "stop"
        toggle GVL.astAxes[Main.hmiAxisSelection].stControl.bStop
    Button (1099,409 124x30), "jogBw", text list: 'languageTable', text index: "jogBw"
        OnMouseDown: execute { GVL.astAxes[Main.hmiAxisSelection].stControl.eCommand:=E_MotionFunctions.eJog; GVL.astAxes[Main.hmiAxisSelection].stControl.bJogBwd:= TRUE; }
        OnMouseClick: execute {  }
        OnMouseUp: execute { GVL.astAxes[Main.hmiAxisSelection].stControl.bJogBwd:= FALSE; }
    Button (1236,409 124x30), "jogFw", text list: 'languageTable', text index: "jogFw"
        OnMouseDown: execute { GVL.astAxes[Main.hmiAxisSelection].stControl.eCommand:=E_MotionFunctions.eJog; GVL.astAxes[Main.hmiAxisSelection].stControl.bJogFwd:= TRUE; }
        OnMouseClick: execute {  }
        OnMouseUp: execute { GVL.astAxes[Main.hmiAxisSelection].stControl.bJogFwd:= FALSE; }
    Button (1100,489 124x30), "HomeRefBwd", input disabled if: GVL.astAxes[MAIN.hmiAxisSelection].stStatus.bGeared, text list: 'languageTable', text index: "eHomeToRef_Bwd"
        OnMouseClick: execute {
            GVL.astAxes[Main.hmiAxisSelection].stControl.eCommand:=E_MotionFunctions.eHome;
            GVL.astAxes[Main.hmiAxisSelection].stConfig.eHomeSeq:=E_HomingRoutines.eHomeToRef_Bwd;
            GVL.astAxes[Main.hmiAxisSelection].stControl.bExecute:=TRUE;
        }
    Button (1236,489 124x30), "HomeRefFwd", input disabled if: GVL.astAxes[MAIN.hmiAxisSelection].stStatus.bGeared, text list: 'languageTable', text index: "eHomeToRef_Fwd"
        OnMouseClick: execute {
            GVL.astAxes[Main.hmiAxisSelection].stControl.eCommand:=E_MotionFunctions.eHome;
            GVL.astAxes[Main.hmiAxisSelection].stConfig.eHomeSeq:=E_HomingRoutines.eHomeToRef_Fwd;
            GVL.astAxes[Main.hmiAxisSelection].stControl.bExecute:=TRUE;
        }
    Button (1100,531 124x30), "HomeDirect", input disabled if: GVL.astAxes[MAIN.hmiAxisSelection].stStatus.bGeared, text list: 'languageTable', text index: "eHomeDirect"
        OnMouseClick: execute {
            GVL.astAxes[Main.hmiAxisSelection].stControl.eCommand:=E_MotionFunctions.eHome;
            GVL.astAxes[Main.hmiAxisSelection].stConfig.eHomeSeq:=E_HomingRoutines.eHomeDirect;
            GVL.astAxes[Main.hmiAxisSelection].stControl.bExecute:=TRUE;
        }
    Button (1100,449 124x30), "HomeLimBwd", input disabled if: GVL.astAxes[MAIN.hmiAxisSelection].stStatus.bGeared, text list: 'languageTable', text index: "eHomeToLimit_Bwd"
        OnMouseClick: execute {
            GVL.astAxes[Main.hmiAxisSelection].stControl.eCommand:=E_MotionFunctions.eHome;
            GVL.astAxes[Main.hmiAxisSelection].stConfig.eHomeSeq:=E_HomingRoutines.eHomeToLimit_Bwd;
            GVL.astAxes[Main.hmiAxisSelection].stControl.bExecute:=TRUE;
        }
    Button (1236,449 124x30), "HomeLimFwd", input disabled if: GVL.astAxes[MAIN.hmiAxisSelection].stStatus.bGeared, text list: 'languageTable', text index: "eHomeToLimit_Fwd"
        OnMouseClick: execute {
            GVL.astAxes[Main.hmiAxisSelection].stControl.eCommand:=E_MotionFunctions.eHome;
            GVL.astAxes[Main.hmiAxisSelection].stConfig.eHomeSeq:=E_HomingRoutines.eHomeToLimit_Fwd;
            GVL.astAxes[Main.hmiAxisSelection].stControl.bExecute:=TRUE;
        }
    Textfield (1100,601 124x30), "%2.2f", text variable: GVL.astAxes[MAIN.hmiAxisSelection].stConfig.fHomePosition
        OnMouseClick: write the text variable via Default
    Textfield (1237,601 124x30), "%2.2f", text variable: GVL.astAxes[MAIN.hmiAxisSelection].stConfig.fHomeFinishDistance
        OnMouseClick: write the text variable via Default
    Textfield (1100,571 124x30), "fHomePosition", text list: 'languageTable', text index: "fHomePosition"
    Textfield (1227,571 145x30), "fHomeFinishDistance", text list: 'languageTable', text index: "fHomeFinishDistance"
    Textfield (239,631 117x30), "bBwEnabled", text list: 'languageTable', text index: "bBwEnabled"
    Lamp1 (209,452 30x30), variable: GVL.astAxes[1].stStatus.bEnabled, style: Lamp-Lamp1-Green
    Textfield (239,452 117x30), "bEnabled", text list: 'languageTable', text index: "bEnabled"
    Lamp1 (209,482 30x30), variable: GVL.astAxes[1].stStatus.bCommandAborted, style: Lamp-Lamp1-Yellow
    Textfield (239,482 117x30), "bCommandAborted", text list: 'languageTable', text index: "bCommandAborted"
    Textfield (239,512 117x30), "bBusy", text list: 'languageTable', text index: "bBusy"
    Lamp1 (209,542 30x30), variable: GVL.astAxes[1].stStatus.bDone, style: Lamp-Lamp1-Green
    Textfield (239,542 117x30), "bDone", text list: 'languageTable', text index: "bDone"
    Lamp1 (209,571 30x30), variable: GVL.astAxes[1].stStatus.bHomed, style: Lamp-Lamp1-Green
    Textfield (239,571 117x30), "bHomed", text list: 'languageTable', text index: "bHomed"
    Lamp1 (209,601 30x30), variable: GVL.astAxes[1].stStatus.bFwEnabled AND NOT GVL.astAxes[1].stStatus.bInterlockedFwd, style: Lamp-Lamp1-Green
    Lamp1 (209,631 30x30), variable: GVL.astAxes[1].stStatus.bBwEnabled AND NOT GVL.astAxes[1].stStatus.bInterlockedBwd, style: Lamp-Lamp1-Green
    Textfield (239,601 117x30), "bFwEnabled", text list: 'languageTable', text index: "bFwEnabled"
    Lamp1 (208,513 30x30), variable: GVL.astAxes[1].stStatus.bBusy, style: Lamp-Lamp1-Yellow
    Textfield (421,33 70x30), "%2.2f", text variable: GVL.astAxes[2].stStatus.fActPosition
    Textfield (366,63 54x30), "actVel", text list: 'languageTable', text index: "actVelocity"
    Textfield (421,63 70x30), "%2.2f", text variable: GVL.astAxes[2].stStatus.fActVelocity
    Textfield (392,631 117x30), "bBwEnabled", text list: 'languageTable', text index: "bBwEnabled"
    Lamp1 (362,452 30x30), variable: GVL.astAxes[2].stStatus.bEnabled, style: Lamp-Lamp1-Green
    Textfield (392,452 117x30), "bEnabled", text list: 'languageTable', text index: "bEnabled"
    Lamp1 (362,482 30x30), variable: GVL.astAxes[2].stStatus.bCommandAborted, style: Lamp-Lamp1-Yellow
    Textfield (392,482 117x30), "bCommandAborted", text list: 'languageTable', text index: "bCommandAborted"
    Textfield (392,512 117x30), "bBusy", text list: 'languageTable', text index: "bBusy"
    Lamp1 (362,542 30x30), variable: GVL.astAxes[2].stStatus.bDone, style: Lamp-Lamp1-Green
    Textfield (392,542 117x30), "bDone", text list: 'languageTable', text index: "bDone"
    Lamp1 (362,571 30x30), variable: GVL.astAxes[2].stStatus.bHomed, style: Lamp-Lamp1-Green
    Textfield (392,571 117x30), "bHomed", text list: 'languageTable', text index: "bHomed"
    Lamp1 (362,601 30x30), variable: GVL.astAxes[2].stStatus.bFwEnabled AND NOT GVL.astAxes[2].stStatus.bInterlockedFwd, style: Lamp-Lamp1-Green
    Lamp1 (362,631 30x30), variable: GVL.astAxes[2].stStatus.bBwEnabled AND NOT GVL.astAxes[2].stStatus.bInterlockedBwd, style: Lamp-Lamp1-Green
    Textfield (392,601 117x30), "bFwEnabled", text list: 'languageTable', text index: "bFwEnabled"
    Lamp1 (361,513 30x30), variable: GVL.astAxes[2].stStatus.bBusy, style: Lamp-Lamp1-Yellow
    Button (926,385 131x30), "reset", pressed state: GVL.astAxes[Main.hmiAxisSelection].stControl.bReset, text list: 'languageTable', text index: "reset"
        OnMouseClick: toggle GVL.astAxes[Main.hmiAxisSelection].stControl.bReset
    Button (1236,531 124x30), "HOME", input disabled if: GVL.astAxes[MAIN.hmiAxisSelection].stStatus.bGeared, text list: 'languageTable', text index: "eHomeDirect"
        OnMouseClick: execute { GVL.astAxes[Main.hmiAxisSelection].stControl.eCommand:=E_MotionFunctions.eHome; GVL.astAxes[Main.hmiAxisSelection].stControl.bExecute:=TRUE; }
    Button (1236,348 124x50), "halt", pressed state: GVL.astAxes[Main.hmiAxisSelection].stControl.bHalt, input disabled if: GVL.astAxes[MAIN.hmiAxisSelection].stStatus.bGeared, text list: 'languageTable', text index: "halt"
        toggle GVL.astAxes[Main.hmiAxisSelection].stControl.bHalt
    Textfield (923,113 57x26), "Enable", text list: 'languageTable', text index: "enable"
    PowerSwitch (922,136 48x48), variable: GVL.astAxes[MAIN.hmiAxisSelection].stControl.bEnable, behaviour: TOGGLE, style: Switch-PowerSwitch-Green
    GroupBox (1224,131 151x150), "Manual Control"
    Button (91,249 87x30), "bLSSOpen"
        toggle LightShutterSystemStates.bLSSOpen
    Lamp1 (47,244 40x39), variable: LightShutterSystemStates.bLSSOpen, style: Lamp-Lamp1-Green
    Button (398,267 98x30), "OPEN - HI", pressed state: LightShutterSystemStates.aOpenToOpen[2]
        toggle LightShutterSystemStates.aOpenToOpen[2]
        OnMouseDown: execute {
            //MAIN.hmiAxisSelection := 2;
            GVL_APP.aLightShutters[2].curPosNbr:=2;
        }
    Textfield (305,362 44x30), "errID", text list: 'languageTable', text index: "errID"
    Textfield (416,97 82x26), "Jog Up/Down", text list: 'languageTable', text index: "jogUpDown"
    Image (423,119 32x32), image: VisuSymbols.Symbols.ArrowBoldUp
        OnMouseDown: execute { LightShutterSystemStates.aJogF[2] := TRUE; }
        OnMouseUp: execute { LightShutterSystemStates.aJogF[2] := FALSE; }
    Image (460,122 32x32), image: VisuSymbols.Symbols.ArrowBoldDown
        OnMouseDown: execute { LightShutterSystemStates.aJogB[2] := TRUE; }
        OnMouseUp: execute { LightShutterSystemStates.aJogB[2] := FALSE; }
    GroupBox (521,187 201x111), "Disable Beamline Operation"
        Button (58,23 113x30), "MIRACLES"
            OnMouseDown: execute { LightShutterSystemStates.aDisabled[1] := NOT(LightShutterSystemStates.aDisabled[1]); }
        Lamp1 (22,23 43x30), variable: LightShutterSystemStates.aDisabled[1], style: Lamp-Lamp1-Red
        Lamp1 (22,61 43x30), variable: LightShutterSystemStates.aDisabled[2], style: Lamp-Lamp1-Red
    Button (579,248 113x30), "HEIMDAL"
        OnMouseDown: execute { LightShutterSystemStates.aDisabled[2] := NOT(LightShutterSystemStates.aDisabled[2]); }
    GroupBox (33,296 150x291), "LSS States"
    RadioButton (45,313 131x266), variable: LightShutterSystemStates.eLightShutterSystemState
        Areas[1]: Text=Closed Off
        Areas[2]: Text=Closed Standby
        Areas[3]: Text=Opening
        Areas[4]: Text=Open
        Areas[5]: Text=Open To Open
        Areas[6]: Text=Adjusting
        Areas[7]: Text=Reset Zero
        Areas[8]: Text=Closing
    Lamp1 (43,603 47x49), variable: LightShutterSystemStates.bPSSPower, style: Lamp-Lamp1-Yellow
    Label (80,602 116x55), "PSS Permission Servo Drives Powered"
    Label (537,133 150x64), "Hide this and think about how it is to be accessed"
    Textfield (458,362 44x30), "errID", text list: 'languageTable', text index: "errID"
    Lamp1 (468,175 30x30), variable: NOT(GVL.astAxes[2].stInputs.bLimitBwd), style: Lamp-Lamp1-Yellow
    Lamp1 (438,175 30x30), variable: NOT(GVL.astAxes[2].stInputs.bLimitBwd), style: Lamp-Lamp1-Yellow
    Label (364,193 45x30), "LSS"
    Label (444,193 45x30), "PSS"
    Label (37,642 173x144), "To do: *Transitions when aborting *Fault state *Torque Homing"
END_VISUALIZATION

// ---- VISUs/languageTable.TcTLO
TEXTLIST languageTable
  axesAvailable = 'PLC Axes available: %d' | Test: 'Alt language'
  velocity = 'Velocity:'
  actposition = 'Position:'
  enable = 'Enable'
  enFW = 'Fwd Enable'
  enBW = 'Bwd Enable'
  axisSel = 'Axis Selected:'
  actVelocity = 'Velocity:'
  errID = 'Error ID:'
  bEnabled = 'Axis Enabled'
  bCommandAborted = 'Command Aborted'
  bBusy = 'Busy'
  bDone = 'Command Done'
  bResetDone = 'Reset Complete'
  bHomed = 'Calibrated'
  bFwEnabled = 'Fwd move enabled'
  bBwEnabled = 'Bwd move enabled'
  bError = 'Error'
  fVelocity = 'Target Vel:'
  fAcceleration = 'Target Acc:'
  fDeceleration = 'Target Dec:'
  fPosition = 'Target Pos:'
  moveAbsolute = 'Abs. pos. move'
  toggle = 'Toggle'
  moveVelocity = 'Const. vel. move'
  bExecute = 'Motion function executed'
  moveRelative = 'Rel. pos. move'
  moveModulo = 'Modulo position move'
  reset = 'Reset axis'
  stop = 'Stop motion'
  jogBw = 'Jog Backward'
  jogFw = 'Jog Forward'
  bGeared = 'In Gear'
  masterGear = 'Master Axis'
  gearRatio = 'Gear Ratio'
  gearIn = 'Gear In'
  gearOut = 'Gear Out'
  eHomeToLimit_Bwd = 'Bwd Limit'
  eHomeToLimit_Fwd = 'Fwd Limit'
  eHomeToRef_Bwd = 'Home Switch Bwd '
  eHomeToRef_Fwd = 'Home Switch Fwd '
  eHomeToEncPulse_Bwd = 'Enc Pulse Bwd '
  eHomeToEncPulse_Fwd = 'Enc Pulse Fwd'
  eHomeToEncPulse_viaBwdLimit = 'EncPulseViaBwdLim'
  eHomeToEncPulse_viaFwdLimit = 'EncPulseViaFwdLim'
  eHomeDirect = 'Home Direct'
  fHomePosition = 'Set Pos after Homing'
  fHomeFinishDistance = 'Rel. Move after Homing'
  halt = 'Halt Motion'
  bInterlockBwd = 'Interlock Bwd'
  bInterlockFwd = 'Interlock Fwd'
  jogUpDown = 'Jog Up/Down'
   = ''
END_TEXTLIST

